(* IEC 61131-3 sources: SCLTeamCoder/experiment/datasets/oscat/oscat_code (part 4) *)

(* ---- FT_IMP.st ---- *)
FUNCTION_BLOCK FT_IMP
VAR_INPUT
    in : REAL;
    T : TIME;
    K : REAL := 1.0;
END_VAR

VAR_OUTPUT
    out : REAL;
END_VAR

VAR
    t1 : FT_PT1;
END_VAR
T1(in:= in, T:=T);
out := (in - t1.out) * K;

(*
hm 3.1.2007	rev 1.1
	added factor K

*)
END_FUNCTION_BLOCK

(* ---- FT_INT.st ---- *)
FUNCTION_BLOCK FT_INT
VAR_INPUT
    IN : REAL;
    K : REAL := 1;
    RUN : BOOL := TRUE;
    RST : BOOL;
    OUT_MIN : REAL := -1E+37;
    OUT_MAX : REAL := 1E+37;
END_VAR

VAR_OUTPUT
    OUT : REAL;
    LIM : BOOL;
END_VAR

VAR
    INTeg : INTEGRATE;
END_VAR
IF rst THEN
	out := 0.0;
ELSE
	integ(X := IN, E := RUN, K := K, Y := out);
END_IF;

(* limit the outputs *)
IF out >= OUT_MAX THEN
	out := out_max;
	LIM := TRUE;
ELSIF out <= out_min THEN
	out := out_min;
	lim := TRUE;
ELSE
	lim := FALSE;
END_IF;

(*
hm 13.12.2006	rev 1.1
	changed to "trapezregel" which increases accuracy
	before out := out + in * time new: out := out + (in + in_last) / 2 * time

hm 15.1.2007		rev 1.2
	added default for k to be 1.

hm	15.9.2007		rev 1.3
	replaced time() with T_PLC_US for compatibility and performance reason
	increased internal accuracy to microseconds

hm 29. oct 2007		rev 1.4
	changed code so int will not be called is time difference is 0 to increase accuracy on systems
	with cycle times below 1ms

hm	2. dec 2007	 	rev 1.5
	changed code for better performance

hm	5. jan 2008		rev 1.6
	further improvements in performance

hm	8. feb 2008		rev 1.7
	deleted limits +/- 1000 now limit is the range of real
	added variables out1 and out2 to extend the resolution
	corrected an error with elapsed time
	deleted unusfull output ET

hm	13. mar 2008	rev 1.8
	changed preset value out_min to -1e37.
	stop integrator at the limits.

hm	16. mar 2008	rev 1.9
	added type conversion to avoid warning under codesys 3.0

hm	2. jun. 2008	rev 2.0
	rewritten with clear code
	limits can now be set without run

hm	3. nov. 2008	rev 2.1
	optimized code using INTEGRATE and LIMX

hm	10. mar. 2009	rev 2.2
	removed nested comments
*)
END_FUNCTION_BLOCK

(* ---- FT_INT2.st ---- *)
FUNCTION_BLOCK FT_INT2
VAR_INPUT
    IN : REAL;
    K : REAL := 1.0;
    RUN : BOOL := TRUE;
    RST : BOOL;
    OUT_MIN : REAL := -1E+38;
    OUT_MAX : REAL := 1E+38;
END_VAR

VAR_OUTPUT
    OUT : REAL;
    LIM : BOOL;
END_VAR

VAR
    integ : INTEGRATE;
    ix : REAL;
    val : REAL2;
END_VAR
IF RST THEN
	val := R2_SET(0.0);
	out := 0.0;
ELSE
	integ(X := IN, E := RUN, K := K, Y := ix);
	val := R2_ADD(val, ix);
	ix := 0.0;
	OUT := val.RX;
END_IF;

(* check output for limits *)
IF out > OUT_MIN AND out < OUT_MAX THEN
	LIM := FALSE;
ELSE
	OUT := LIMIT(OUT_MIN, OUT, OUT_MAX);
	val := R2_SET(OUT);
	LIM := TRUE;
END_IF;

(*	revision history
hm	2. jun. 2008	rev 1.0
	original version

hm	5. nov. 2008	rev 1.1
	rewritten code using integrate

hm	11. mar. 2009	rev 1.2
	real constants updated to new systax using dot

*)
END_FUNCTION_BLOCK

(* ---- FT_MIN_MAX.st ---- *)
FUNCTION_BLOCK FT_MIN_MAX
VAR_INPUT
    in : REAL;
    rst : BOOL;
END_VAR

VAR_OUTPUT
    mx : REAL;
    mn : REAL;
END_VAR

VAR
    init : BOOL;
END_VAR
IF rst OR NOT init THEN
	mn := in;
	mx := in;
	init := TRUE;
ELSIF in < mn THEN mn := in;
ELSIF in > mx THEN mx := in;
END_IF;
END_FUNCTION_BLOCK

(* ---- FT_PD.st ---- *)
FUNCTION_BLOCK FT_PD
VAR_INPUT
    IN : REAL;
    KP : REAL := 1.0;
    TV : REAL := 1.0;
END_VAR

VAR_OUTPUT
    Y : REAL;
END_VAR

VAR
    diff : FT_DERIV;
END_VAR
(* run differentiator *)
diff(IN := IN, K := TV);

(* combine both values *)
Y := KP * (diff.out + IN);

(* revision history
hm 	3. jun. 2008 	rev 1.0
	original version

*)
END_FUNCTION_BLOCK

(* ---- FT_PDT1.st ---- *)
FUNCTION_BLOCK FT_PDT1
VAR_INPUT
    IN : REAL;
    KP : REAL := 1.0;
    TV : REAL := 1.0;
    T1 : REAL := 1.0;
END_VAR

VAR_OUTPUT
    Y : REAL;
END_VAR

VAR
    diff : FT_DERIV;
    TP : FT_PT1;
END_VAR
(* run differentiator *)
diff(IN := IN, K := TV);

(* Run PT1 filter *)
tp(in := diff.out, T := REAL_TO_TIME(T1));

(* combine both values *)
Y := KP * (tp.out + IN);

(* revision history
hm 	3. jun. 2008 	rev 1.0
	original version

*)
END_FUNCTION_BLOCK

(* ---- FT_PI.st ---- *)
FUNCTION_BLOCK FT_PI
VAR_IN
    IN : REAL;
    KP : REAL := 1.0;
    KI : REAL := 1.0;
    ILIM_L : REAL := -1E+38;
    ILIM_H : REAL := 1E+38;
    IEN : BOOL := TRUE;
    RST : BOOL;
END_VAR

VAR_OUT
    Y : REAL;
    LIM : BOOL;
END_VAR

VAR
    integ : FT_INT;
END_VAR
(* run integrator *)
integ(IN := IN, K := KI, RUN := IEN, RST := RST, OUT_MIN := ILIM_L, OUT_MAX := ILIM_H);

(* check if integrator has reached its limits and set overflow *)
LIM := integ.LIM;
Y := KP * IN + integ.Out;

(* revision history
hm 	3. jun. 2008 	rev 2.0
	original version

*)
END_FUNCTION_BLOCK

(* ---- FT_PID.st ---- *)
FUNCTION_BLOCK FT_PID
VAR_INPUT
    IN : REAL;
    KP : REAL := 1.0;
    TN : REAL := 1.0;
    TV : REAL := 1.0;
    ILIM_L : REAL := -1E+38;
    ILIM_H : REAL := 1E+38;
    IEN : BOOL := TRUE;
    RST : BOOL;
END_VAR

VAR_OUTPUT
    Y : REAL;
    LIM : BOOL;
END_VAR

VAR
    integ : FT_INT;
    diff : FT_DERIV;
END_VAR
(* run integrator only if TN > 0 *)
IF TN > 0.0 THEN
	integ(IN := IN, K := 1.0 / TN, RUN := IEN, RST := RST, OUT_MIN := ILIM_L, OUT_MAX := ILIM_H);
ELSE
	integ(RST := FALSE);
END_IF;

(* run differentiator *)
diff(IN := IN, K := TV);

(* combine both values *)
Y := KP * (integ.Out + diff.out + IN);

(* check if integrator has reached its limits and set overflow *)
LIM := integ.LIM;

(* revision history
hm 3. jun. 2008 	rev 2.0
	original version

hm	11. mar. 2009	rev 2.1
	real constants updated to new systax using dot

*)
END_FUNCTION_BLOCK

(* ---- FT_PIDW.st ---- *)
FUNCTION_BLOCK FT_PIDW
VAR_INPUT
    IN : REAL;
    KP : REAL := 1.0;
    TN : REAL := 1.0;
    TV : REAL := 1.0;
    LIM_L : REAL := -1E+38;
    LIM_H : REAL := 1E+38;
    RST : BOOL;
END_VAR

VAR_OUTPUT
    Y : REAL;
    LIM : BOOL;
END_VAR

VAR
    integ : INTEGRATE;
    diff : FT_DERIV;
    YI : REAL;
END_VAR
(* run the integrator *)
IF tn = 0.0 OR rst THEN
	integ(E := FALSE, Y := YI);
	YI := 0.0;
ELSE
	integ(X := IN, K := 1.0 / TN, E := NOT LIM, Y := YI);
END_IF;

(* add up integrator and linear part *)
Y := KP * (IN + YI);

(* run differentiator *)
diff(IN := IN, K := TV);

(* set lim before differentiator is added to stop integrator if necessary *)
IF Y > LIM_L AND Y < LIM_H THEN
	LIM := FALSE;
ELSE
	LIM := TRUE;
END_IF;

(* add differential part and limit output Y *)

Y := LIMIT(LIM_L, Y + KP * diff.out, LIM_H);

(* revision history
hm 3. jun. 2008 	rev 1.0
	original version

hm	5. nov. 2008	rev 1.1
	changed code to use integrate

hm	11. mar. 2009	rev 1.2
	real constants updated to new systax using dot

*)
END_FUNCTION_BLOCK

(* ---- FT_PIDWL.st ---- *)
FUNCTION_BLOCK FT_PIDWL
VAR_INPUT
    IN     : REAL;
    KP     : REAL := 1.0;
    TN     : REAL := 1.0;
    TV     : REAL := 1.0;
    LIM_L  : REAL := -1E+38;
    LIM_H  : REAL := 1E+38;
    RST    : BOOL;
END_VAR

VAR_OUTPUT
    Y      : REAL;
    LIM    : BOOL;
END_VAR

VAR
    piwl   : FT_PIWL; // derived type
    diff   : FT_DERIV; // derived type
END_VAR
(* if rst then *)
IF rst THEN
	piwl(rst := TRUE);
	piwl.RST := FALSE;
ELSE
	(* run PIWL controller first *)
	(* we need to check if TN = 0 and do alternative calls *)
	IF TN = 0.0 THEN
		piwl(in := IN * KP, KP := 1.0, KI := 0.0, LIM_L := LIM_L, LIM_H := LIM_H);
	ELSE
		piwl(in := IN * KP, KP := 1.0, KI := 1.0 / TN, LIM_L := LIM_L, LIM_H := LIM_H);
	END_IF;

	(* run differentiator and add_to_output *)
	diff(IN := IN, K := KP * TV);
	Y := piwl.Y + diff.out;

	(* limit the output *)
	IF Y < LIM_L THEN
		LIM := TRUE;
		Y := LIM_L;
	ELSIF Y > LIM_H THEN
		LIM := TRUE;
		Y := LIM_H;
	ELSE
		LIM := FALSE;
	END_IF;
END_IF;

(* revision history
hm 13. jun. 2008 	rev 1.0
	original version

hm	25. jan 2008	rev 1.1
	multiply differential part with KP

hm	11. mar. 2009	rev 1.2
	real constants updated to new systax using dot

hm	13. nov. 2009	rev 1.3
	fixed code for negative KP

*)
END_FUNCTION_BLOCK

(* ---- FT_PIW.st ---- *)
FUNCTION_BLOCK FT_PIW
VAR_INPUT
    IN : REAL;
    KP : REAL := 1.0;
    KI : REAL := 1.0;
    LIM_L : REAL := -1E+38;
    LIM_H : REAL := 1E+38;
    RST : BOOL;
END_VAR

VAR_OUTPUT
    Y : REAL;
    LIM : BOOL;
END_VAR

VAR
    integ : FT_INT;
END_VAR
(* run integrator *)
integ(IN := IN, K := KI, RUN := NOT LIM, RST := RST);

(* set output value *)
Y := KP * IN + integ.Out;

(* check for limits and set integrator for anti wind up *)
IF Y < LIM_L THEN
	Y := LIM_L;
	LIM := TRUE;
ELSIF Y > LIM_H THEN
	Y := LIM_H;
	LIM := TRUE;
ELSE
	LIM := FALSE;
END_IF;

(* revision history
hm 	3. jun. 2008 	rev 1.0
	original version

*)
END_FUNCTION_BLOCK

(* ---- FT_PIWL.st ---- *)
FUNCTION_BLOCK FT_PIWL
VAR_INPUT
    IN : REAL;
    KP : REAL := 1.0;
    KI : REAL := 1.0;
    LIM_L : REAL := -1E+38;
    LIM_H : REAL := 1E+38;
    RST : BOOL;
END_VAR

VAR_OUTPUT
    Y : REAL;
    LIM : BOOL;
END_VAR

VAR
    init : BOOL;
    tx : DWORD;
    tc : REAL;
    t_last : DWORD;
    in_last : REAL;
    i : REAL;
    p : REAL;
END_VAR
(* initialize at power_up *)
IF NOT init OR RST THEN
	init := TRUE;
	in_last := in;
	t_last := T_PLC_US();
	i := 0.0;
	tc := 0.0;
ELSE
	(* read last cycle time in Microseconds *)
	tx := T_PLC_US();
	tc := DWORD_TO_REAL(tx - t_last);
	t_last := tx;

	(* calculate proportional part *)
	p := KP * IN;

	(* run integrator *)
	i := (IN + in_last) * 5.0E-7 * KI * tc + i;
	in_last := IN;

	(* calculate output Y *)
	Y := p + i;

	(* check output for limits *)
	IF Y >= LIM_H THEN
		Y := LIM_H;
		IF ki <> 0.0 THEN
			i := LIM_H - p;
		ELSE
			i := 0.0;
		END_IF;
		LIM := TRUE;
	ELSIF Y <= LIM_L THEN
		Y := LIM_L;
		IF ki <> 0.0 THEN
			i := LIM_L - p;
		ELSE
			i := 0.0;
		END_IF;
		LIM := TRUE;
	ELSE
		LIM := FALSE;
	END_IF;
END_IF;

(* revision history
hm 13. jun. 2008 	rev 1.0
	original version

hm	27. oct. 2008	rev 1.1
	integrator will not be adjusted when ki = 0

hm	25. jan 2009	rev 1.2
	module will also work with negative K

hm	11. mar. 2009	rev 1.3
	real constants updated to new systax using dot

*)
END_FUNCTION_BLOCK

(* ---- FT_Profile.st ---- *)
FUNCTION_BLOCK FT_Profile
VAR_INPUT
    K : REAL := 1.0;
    O : REAL;
    M : REAL := 1.0;
    E : BOOL;
    value_0 : REAL;
    time_1 : TIME;
    value_1 : REAL;
    time_2 : TIME;
    value_2 : REAL;
    time_3 : TIME;
    value_3 : REAL;
    time_10 : TIME;
    value_10 : REAL;
    time_11 : TIME;
    value_11 : REAL;
    time_12 : TIME;
    value_12 : REAL;
    time_13 : TIME;
    value_13 : REAL;
END_VAR_INPUT

VAR_OUTPUT
    Y : REAL;
    RUN : BOOL;
    ET : TIME;
END_VAR_OUTPUT

VAR
    tx : TIME;
    edge : BOOL;
    state : BYTE;
    ta : TIME;
    tb : TIME;
    t0 : TIME;
    temp : REAL;
    va : REAL;
    vb : REAL;
END_VAR
(* read system time *)
tx := DWORD_TO_TIME(T_PLC_MS());

(* determine start condition *)
IF E AND NOT edge THEN
	RUN := TRUE;
	ET := t#0s;
	t0 := tx;
	ta := tx;
	tb := multime(time_1, M);
	va := value_0;
	vb := value_1;
	temp := value_0;
	state := 1;
END_IF;
edge := E;

(* generate startup profile *)
IF run THEN
	CASE state OF
		1:	IF tx - ta >= tb THEN
				ta := ta + tb;
				tb := multime(time_2 - time_1, M);
				va := value_1;
				vb := value_2;
				temp := value_1;
				state := 2;
			ELSE
				temp := ((vb - va) * TIME_TO_REAL(tx - ta) / TIME_TO_REAL(tb) + va);
			END_IF;
		2:	IF tx - ta >= tb THEN
				ta := ta + tb;
				tb := multime(time_3 - time_2, M);
				va := value_2;
				vb := value_3;
				temp := value_2;
				state := 3;
			ELSE
				temp := ((vb - va) * TIME_TO_REAL(tx - ta) / TIME_TO_REAL(tb) + va);
			END_IF;
		3:	IF tx - ta >= tb THEN
				ta := ta + tb;
				tb := multime(time_10 - time_3, M);
				va := value_3;
				vb := value_10;
				temp := value_3;
				state := 4;
			ELSE
				temp := ((vb - va) * TIME_TO_REAL(tx - ta) / TIME_TO_REAL(tb) + va);
			END_IF;
		4 :	IF tx - ta >= tb THEN
				ta := ta + tb;
				tb := multime(time_11 - time_10, M);
				va := value_10;
				vb := value_11;
				temp := value_10;
				IF E THEN state := 5; ELSE state := 6; END_IF;
			ELSE
				temp := ((vb - va) * TIME_TO_REAL(tx - ta) / TIME_TO_REAL(tb) + va);
			END_IF;
		5:	(* extend the signal while E is true *)
			IF E THEN
				ta := tx;
			ELSE
				state := 6;
			END_IF;
		6:	IF tx - ta >= tb THEN
				ta := ta + tb;
				tb := multime(time_12 - time_11, M);
				va := value_11;
				vb := value_12;
				temp := value_11;
				state := 7;
			ELSE
				temp := ((vb - va) * TIME_TO_REAL(tx - ta) / TIME_TO_REAL(tb) + va);
			END_IF;
		7:	IF tx - ta >= tb THEN
				ta := ta + tb;
				tb := multime(time_13 - time_12, M);
				va := value_12;
				vb := value_13;
				temp := value_12;
				state := 8;
			ELSE
				temp := ((vb - va) * TIME_TO_REAL(tx - ta) / TIME_TO_REAL(tb) + va);
			END_IF;
		8:	IF tx - ta >= tb THEN
				temp := value_13;
				run := FALSE;
			ELSE
				temp := ((vb - va) * TIME_TO_REAL(tx - ta) / TIME_TO_REAL(tb) + va);
			END_IF;
	END_CASE;
	Y := temp * K + O;
	ET := tx - t0;
END_IF;

(* revision history
hm	27 feb 2007		rev 1.0
	original version

hm	15. sep2007		rev 1.1
	replaced Time() with T_PLC_MS for compatibility and performance reasons

*)
END_FUNCTION_BLOCK

(* ---- FT_PT1.st ---- *)
FUNCTION_BLOCK FT_PT1
VAR_INPUT
    in : REAL;
    T : TIME;
    K : REAL := 1.0;
END_VAR

VAR_OUTPUT
    out : REAL;
END_VAR

VAR
    last : DWORD;
    tx : DWORD;
    init : BOOL;
END_VAR
(* read system time *)
tx := T_PLC_US();

(* startup initialisation *)
IF NOT init OR T = t#0s THEN
	init := TRUE;
	out := K * in;
ELSE
	out := out + (in * K - out) * DWORD_TO_REAL(Tx - last) / TIME_TO_REAL(T) * 1.0E-3;
	IF ABS(out) < 1.0E-20 THEN out := 0.0; END_IF;
END_IF;
last := tx;

(*
hm 1.1.2007	rev 1.1
	corrected error while startup value was not correct
	for very small time values real output would run out of range.

hm 3.1.2007	rev 1.2
	corrected an error for falling edge failures.
	added output faktor K.

hm 27. 2. 2007	rev 1.3
	output will be input during init for definitive startup condition.

hm	15.9.2007	rev 1.4
	changed time() to T_PLC_US() for compatibilitxy resons
	increased internal accuracy to Microseconds instead of Milliseconds

hm	23. oct 2007	rev 1.5
	added out := in to the init statements

hm	30. nov 2007	rev 1.6
	changed out to be K * in during initialization

hm	5. jan 2008	rev 1.7
	improved code for better performance

hm	16. mar. 2008	rev 1.8
	added type conversion to avoid warning under codesys 3.0

hm	14. jun. 2008	rev 1.9
	improved code

hm	11. mar. 2009	rev 1.10
	real constants updated to new systax using dot

hm	18. jan. 2011	rev 1.11
	avoid underrun of out
*)
END_FUNCTION_BLOCK

(* ---- FT_PT2.st ---- *)
FUNCTION_BLOCK FT_PT2
VAR_INPUT
    in : REAL;
    T : TIME;
    D : REAL;
    K : REAL := 1.0;
END_VAR

VAR_OUTPUT
    out : REAL;
END_VAR

VAR
    init : BOOL;
    int1 : INTEGRATE;
    int2 : INTEGRATE;
    tn : REAL;
    I1 : REAL;
    I2 : REAL;
    tn2 : REAL;
END_VAR
(* startup initialisation *)
IF NOT init OR T = T#0s THEN
	init := TRUE;
	out := K * in;
	I2 := out;
ELSE
	TN := TIME_TO_REAL(T) * 1.0E-3;
	tn2 := TN * TN;
	int1(X := in * K / tn2 - I1 * 0.5 * D / TN - I2 / TN2, Y := I1);
	int2(X := I1,Y := I2);
	out := I2;
END_IF;

(* revision history

15.1.2007 hm		rev 1.1
	changed formula to new more acurate formula

hm 15.9.2007		rev 1.2
	deleted unused code for init system time reading tx

hm	30.11.2007	rev 1.3
	changed out to be K * in during initialization
	avoind divide by 0 if tn = 0

hm	3. nov. 2008	rev 1.4
	optimized code and fixed a problem with init

hm	11. mar. 2009	rev 1.5
	real constants updated to new systax using dot

*)
END_FUNCTION_BLOCK

(* ---- FT_RMP.st ---- *)
FUNCTION_BLOCK FT_RMP
VAR_INPUT
    Rmp : BOOL := TRUE;
    in : REAL;
    KR : REAL;
    KF : REAL;
END_VAR

VAR_OUTPUT
    out : REAL;
    busy : BOOL;
    UD : BOOL;
END_VAR

VAR
    tx : TIME;
    last : TIME;
    init : BOOL;
END_VAR
(* read system time *)
tx := DWORD_TO_TIME(T_PLC_MS()) - last;

IF NOT init THEN
	init := TRUE;
	last := tx;
	tx := t#0s;
	out := in;
END_IF;
IF NOT rmp THEN
	out := in;
	busy := FALSE;
ELSIF out > in THEN
	(* ramp down *)
	out := out - TIME_TO_REAL(tx) * 0.001 * KF;
	out := MAX(in, out);
ELSIF out < in THEN
	(* ramp up *)
	out := out + TIME_TO_REAL(tx) * 0.001 * KR;
	out := MIN(in, out);
END_IF;

(* set busy and dir flags *)
IF out < in THEN
	busy := TRUE;
	ud := TRUE;
ELSIF out > in THEN
	busy := TRUE;
	ud := FALSE;
ELSE
	busy := FALSE;
END_IF;
last := last + tx;

(* revision history:

hm 8.10.2006			rev 1.1
	added ud output

hm 12. feb 2007		rev 1.2
	added init variable and corrected a possible startup problem

hm	17. sep 2007	rev 1.3
	replaced time() with t_plc_ms() for compatibility reasons

hm	25. jan 2008	rev 1.4
	performance improvements
	allow KR and KF to be 0
*)
END_FUNCTION_BLOCK

(* ---- FT_TN16.st ---- *)
FUNCTION_BLOCK FT_TN16
VAR_INPUT
    in : REAL;
    T : TIME;
END_VAR

VAR_OUTPUT
    out : REAL;
    trig : BOOL;
END_VAR

VAR
    length : INT := 16;
    X : ARRAY[0..15] OF REAL;
    cnt : INT;
    last : TIME;
    tx : TIME;
    init : BOOL;
END_VAR
(* read system time *)
tx := DWORD_TO_TIME(T_PLC_MS());

trig := FALSE;
IF NOT init THEN
	x[cnt] := in;
	init := TRUE;
	last := tx;
ELSIF tx - last >= T / length THEN
	IF cnt = length - 1 THEN cnt := 0; ELSE cnt := cnt + 1; END_IF;
	Out := X[cnt];
	x[cnt] := in;
	last := tx;
	Trig := TRUE;
END_IF;

(* revision history
hm		1. jan 2007	rev 1.0
	original version

hm		16. sep 2007	rev 1.1
	changes time() to T_plc_ms() for compatibility reasons

*)
END_FUNCTION_BLOCK

(* ---- FT_TN64.st ---- *)
FUNCTION_BLOCK FT_TN64
VAR_INPUT
    in: REAL;
    T: TIME;
END_VAR

VAR_OUTPUT
    out: REAL;
    trig: BOOL;
END_VAR

VAR
    length: INT := 64;
    X: ARRAY[0..63] OF REAL;
    cnt: INT;
    last: TIME;
    tx: TIME;
    init: BOOL;
END_VAR
(* read system time *)
tx := DWORD_TO_TIME(T_PLC_MS());

trig := FALSE;
IF NOT init THEN
	x[cnt] := in;
	init := TRUE;
	last := tx;
ELSIF tx - last >= T / length THEN
	IF cnt = length - 1 THEN cnt := 0; ELSE cnt := cnt + 1; END_IF;
	Out := X[cnt];
	x[cnt] := in;
	last := tx;
	trig := TRUE;
END_IF;

(* revision history
hm		1. jan 2007		rev 1.0
	original version

hm		16. sep 2007	rev 1.1
	changes time() to T_plc_ms() for compatibility reasons

*)
END_FUNCTION_BLOCK

(* ---- FT_TN8.st ---- *)
FUNCTION_BLOCK FT_TN8
VAR_INPUT
    in : REAL;
    T : TIME;
END_VAR

VAR_OUTPUT
    out : REAL;
    trig : BOOL;
END_VAR

VAR
    length : INT := 8;
    X : ARRAY[0..7] OF REAL;
    cnt : INT;
    last : TIME;
    tx : TIME;
    init : BOOL;
END_VAR
tx := DWORD_TO_TIME(T_PLC_MS());
trig := FALSE;
IF NOT init THEN
	x[cnt] := in;
	init := TRUE;
	last := tx;
ELSIF tx - last >= T / length THEN
	IF cnt = length - 1 THEN cnt := 0; ELSE cnt := cnt + 1; END_IF;
	Out := X[cnt];
	x[cnt] := in;
	last := tx;
	trig := TRUE;
END_IF;

(* revision history
hm		1. jan 2007		rev 1.0
	original version

hm		16. sep 2007	rev 1.1
	changes time() to T_plc_ms() for compatibility reasons

*)
END_FUNCTION_BLOCK

(* ---- GEN_BIT.st ---- *)
FUNCTION_BLOCK GEN_BIT
VAR_INPUT
    in0 : DWORD;
    in1 : DWORD;
    in2 : DWORD;
    in3 : DWORD;
    clk : BOOL;
    steps : INT;
    rep : INT;
    rst : BOOL;
END_VAR

VAR_OUTPUT
    Q0 : BOOL;
    Q1 : BOOL;
    Q2 : BOOL;
    Q3 : BOOL;
    cnt : INT;
    run : BOOL;
END_VAR

VAR
    r0 : DWORD;
    r1 : DWORD;
    r2 : DWORD;
    r3 : DWORD;
    rx : INT := 1;
END_VAR
(* check if number of runs is finished or rep = 0 which means continuous *)

IF clk AND NOT rst THEN
	run := (rep = 0) OR (rx <= rep);
	IF run THEN
		(* check for step counter reached and reset to 0 if cnt = steps *)
		IF cnt = steps THEN
			cnt := 0;
		END_IF;

		(* when cnt = 0 then reload the inputs into the registers *)
		IF cnt = 0 THEN
			r0 := in0;
			r1 := in1;
			r2 := in2;
			r3 := in3;
		END_IF;

		(* when cnt < steps, shift the lowest bits to the outputs *)
		IF (cnt < steps) THEN
			Q0 := r0.0;
			Q1 := r1.0;
			Q2 := r2.0;
			Q3 := r3.0;
			r0 := SHR(r0,1);
			r1 := SHR(r1,1);
			r2 := SHR(r2,1);
			r3 := SHR(r3,1);
		END_IF;

		(* increment the step counter *)
		cnt := cnt +1;
		IF (cnt = steps) AND (rep <> 0) THEN rx := rx +1; END_IF;
		IF (rx > rep) AND (rep <> 0) THEN run := FALSE; END_IF;
	END_IF;
ELSE
	IF rst THEN
		run := FALSE;
		Q0 := FALSE;
		Q1 := FALSE;
		Q2 := FALSE;
		Q3 := FALSE;
		r0 := 0;
		r1 := 0;
		r2 := 0;
		r3 := 0;
		cnt := 0;
		rx := 1;
	END_IF;
END_IF;

(* revision histroy
hm	4 aug 2006	rev 1.0
	original version

hm 15. oct. 2008	rev 1.1
	improved performance

hm	14. mar. 2009	rev 1.2
	removed double assignments

*)
END_FUNCTION_BLOCK

(* ---- GEN_PULSE.st ---- *)
FUNCTION_BLOCK GEN_PULSE
VAR_INPUT
    ENQ : BOOL := TRUE;
    PTH : TIME;
    PTL : TIME;
END_VAR

VAR_OUTPUT
    Q : BOOL;
END_VAR

VAR
    tx : TIME;
    tn : TIME;
    init : BOOL;
END_VAR
IF enq THEN
	tx := DWORD_TO_TIME(T_PLC_MS());
	IF NOT init THEN init := TRUE; tn := tx; END_IF;
	IF tx - tn >= SEL(Q, PTL, PTH) THEN
		tn := tn + SEL(Q, PTL, PTH);
		Q := NOT Q;
	END_IF;
ELSE
	Q := FALSE;
	init := FALSE;
END_IF;

(* revision history
hm	29. jun. 2008	rev 1.0
	original version

hm	23. nov. 2008	rev 1.1
	set default for enq to be true

hm	18. jul. 2009	rev 1.2
	improved performance

hm	13. nov. 2009	rev 1.3
	corrected error

hm	16. feb. 2011	rev 1.4
	corrected an error when timer overflows

hm	8. apr. 2011	rev 1.5
	ptl and pth was exchanged
*)
END_FUNCTION_BLOCK

(* ---- GEN_PW2.st ---- *)
FUNCTION_BLOCK GEN_PW2
VAR_INPUT
    ENQ: BOOL;
    TH1: TIME;
    TL1: TIME;
    TH2: TIME;
    TL2: TIME;
    TS: BOOL;
END_VAR

VAR_OUTPUT
    Q: BOOL;
    TH: TIME;
    TL: TIME;
END_VAR

VAR
    t_high: TIME;
    t_low: TIME;
    tx: TIME;
    start: TIME;
    init: BOOL;
    et: TIME;
END_VAR
(* read system timer *)
tx := DWORD_TO_TIME(T_PLC_MS());

(* startup initialization *)
IF NOT init THEN
	start := tx;
	init := TRUE;
	TH := T#0s;
	TL := T#0s;
END_IF;

(* timing selection *)
IF TS THEN
	t_high := TH2;
	t_low := TL2;
ELSE
	t_high := TH1;
	t_low := TL1;
END_IF;

(* normal operation *)
IF ENQ THEN
	et := tx - start;
	IF NOT Q THEN
		IF et >= t_low THEN
			Q := TRUE;
			start := tx;
			TL := T#0s;
		ELSE
			TL := et;
		END_IF;
	ELSE
		IF et >= t_high THEN
			Q := FALSE;
			start := tx;
			TH := T#0s;
		ELSE
			TH := et;
		END_IF;
	END_IF;
ELSE
	Q := FALSE;
	TH := T#0s;
	TL := T#0s;
	start := tx;
END_IF;

(* revision history
hm	26. sep. 2008	rev 1.0
	original version

hm	14. mar. 2009	rev 1.1
	removed double assignments

*)
END_FUNCTION_BLOCK

(* ---- GEN_RDM.st ---- *)
FUNCTION_BLOCK GEN_RDM
VAR_INPUT
    PT : TIME;
    AM : REAL := 1;
    OS : REAL;
END_VAR

VAR_OUTPUT
    Q : BOOL;
    Out : REAL;
END_VAR

VAR
    tx : TIME;
    last : TIME;
    init : BOOL;
END_VAR
(* read system time and prepare input data *)
tx := DWORD_TO_TIME(T_PLC_MS()) - last;

(* init section *)
IF NOT init THEN
	init := TRUE;
	last := tx;
	tx := t#0s;
END_IF;

(* add last if one cycle is finished *)
IF tx >= pt THEN
	last := last + pt;
	tx := tx - pt;

	(* generate output signal *)
	out := am * (RDM(0) - 0.5) + os;
	q := TRUE;
ELSE
	q := FALSE;
END_IF;

(* revision history

hm	7.2.2007		rev 1.0
	original version

hm	16.9.2007		rev 1.1
	changes time() to T_plc_ms() for compatibility reasons

*)
END_FUNCTION_BLOCK

(* ---- GEN_RDT.st ---- *)
FUNCTION_BLOCK GEN_RDT
VAR_INPUT
    Enable : BOOL := TRUE;
    Min_Time_ms : TIME := TIME#1s0ms; // min Taktzeit
    Max_Time_ms : TIME := TIME#1s200ms; // Max Taktzeit
    TP_Q : TIME := TIME#100ms; // Zeit Ausgang auf TRUE
END_VAR

VAR_OUTPUT
    xQ : BOOL;
END_VAR

VAR
    tonRDMTimer : TON; // Zeitbaustein Taktgenerator
    tof_xQ : TOF; // Ausschaltverzögerung Taktgenerator
    tRDMTime : TIME; // Sollzeit
    rRDMTime : REAL; // Zufalswert Timer
END_VAR
tonRDMTimer ( IN:= Enable , PT:= tRDMTime );
tof_xQ ( IN:= tonRDMTimer.Q , PT:= TP_Q );
XQ := tof_xq.Q;
IF tonRDMTimer.Q THEN
		 xQ := TRUE ;
		 rRDMTime := RDM ( last:= rRDMTime ) ;
		 tRDMTime := REAL_TO_TIME ( rRDMTime * DINT_TO_REAL(TIME_TO_DINT( Max_Time_ms - Min_Time_ms ) + TIME_TO_DINT(Min_Time_ms ))) ;
		 tonRDMTimer ( IN:= FALSE );
END_IF;

(* revision history
J. Schohaus	19. nov 2007	rev 1.0
	origial version

hm	16. mar. 2008			rev 1.1
	added type conversion to avoid warnings under codesys 3.0
*)
END_FUNCTION_BLOCK

(* ---- GEN_RMP.st ---- *)
FUNCTION_BLOCK GEN_RMP
VAR_INPUT
    PT : TIME := TIME#1s0ms;
    AM : REAL := 1.0;
    OS : REAL;
    DL : REAL;
END_VAR

VAR_OUTPUT
    Q : BOOL;
    OUT : REAL;
END_VAR

VAR
    tx : TIME;
    last : TIME;
    init : BOOL;
    temp : REAL;
    ltemp : REAL;
END_VAR
(* read system time and prepare input data *)
tx := DWORD_TO_TIME(T_PLC_MS()) - last;
DL := MODR(dl,1.0);
IF dl < 0.0 THEN dl := 1.0 - dl; END_IF;

(* init section *)
IF NOT init THEN
	init := TRUE;
	last := tx;
	tx := t#0s;
END_IF;

(* add last if one cycle is finished *)
IF tx >= pt THEN
	last := last + pt;
	tx := tx - pt;
END_IF;

(* generate sine wave *)
ltemp := temp;
IF pt > t#0s THEN temp := FRACT(TIME_TO_REAL(tx + MULTIME(pt, dl)) / TIME_TO_REAL(pt)); END_IF;
out := am * temp + os;

(* boolean output Q *)
Q := temp < ltemp;

(* revision history
hm	3. mar 2007		rev 1.0
	original version

hm	17 sep 2007		rev 1.1
	replaced time() with t_plc_ms for compatibilitx reasons

hm	27. nov 2007	rev 1.2
	avoid divide by 0 when pt = 0

ks	26. oct. 2008	rev 1.3
	code optimization

hm	10. mar. 2009	rev 1.4
	changed real constants to use dot syntax
*)
END_FUNCTION_BLOCK

(* ---- GEN_SIN.st ---- *)
FUNCTION_BLOCK GEN_SIN
VAR_INPUT
    PT : TIME;
    AM : REAL := 1.0;
    OS : REAL;
    DL : REAL;
END_VAR

VAR_OUTPUT
    Q : BOOL;
    Out : REAL;
END_VAR

VAR
    tx : TIME;
    last : TIME;
    init : BOOL;
    temp : REAL;
END_VAR
(* read system time and prepare input data *)
tx := DWORD_TO_TIME(T_PLC_MS()) - last;
DL := MODR(dl,1.0);
IF dl < 0.0 THEN dl := 1.0 - dl; END_IF;

(* init section *)
IF NOT init THEN
	init := TRUE;
	last := tx;
	tx := t#0s;
END_IF;

(* add last if one cycle is finished *)
IF tx >= pt THEN
	last := last + pt;
	tx := tx - pt;
END_IF;

(* generate sine wave *)
IF pt > t#0s THEN temp := SIN(math.PI2 * DWORD_TO_REAL(TIME_TO_DWORD(tx + MULTIME(pt, dl))) / DWORD_TO_REAL(TIME_TO_DWORD(pt))); END_IF;
out := am * 0.5 *  temp + os;

(* boolean output Q *)
q := NOT SIGN_R(temp);

(* revision history
hm	22. jan 2007	rev 1.0
	original version

hm	17 sep 2007	rev 1.1
	replaced time() with t_plc_ms for compatibilitx reasons

hm	27. nov 2007	rev 1.2
	avoid divide by 0 when pt = 0

hm	6. jan 2008		rev 1.3
	improved performance

hm	16. mar. 2008	rev 1.4
	added type conversion to avoid warnings under codesys 3.0

hm	18. oct. 2008	rev 1.5
	using math constants

hm	11. mar. 2009	rev 1.6
	changed real constants to use dot syntax

*)
END_FUNCTION_BLOCK

(* ---- GEN_SQ.st ---- *)
FUNCTION_BLOCK GEN_SQ
VAR_INPUT
    PT: TIME;
END_VAR

VAR_OUTPUT
    Q: BOOL;
END_VAR

VAR
    tn: DWORD;
    tx: DWORD;
    init: BOOL;
END_VAR
(* read system time *)
tx := T_PLC_MS();

IF NOT init THEN
	init := TRUE;
	tn := tx;
	Q := TRUE;
ELSIF tx - tn >= SHR(TIME_TO_DWORD(PT),1) THEN
	Q := NOT Q;
	tn := tn + SHR(TIME_TO_DWORD(pt),1);
END_IF;

(* revision history
hm	4. aug 2006	rev 1.0
	original version

hm	17. sep 2007	rev 1.1
	replaced time() with T_PLC_MS() for compatibility reasons

hm	18. jul. 2009	rev 1.2
	improved accuracy

hm	16. feb 2011	rev 1.3
	corrected an error with timer overflow
*)
END_FUNCTION_BLOCK

(* ---- GEN_SQR.st ---- *)
FUNCTION_BLOCK GEN_SQR
VAR_INPUT
    PT : TIME;
    AM : REAL := 1.0;
    OS : REAL;
    DC : REAL := 0.5;
    DL : REAL;
END_VAR

VAR_OUTPUT
    Q : BOOL;
    Out : REAL;
END_VAR

VAR
    tx : TIME;
    last : TIME;
    init : BOOL;
END_VAR
(* check dc = 1 or 0 *)
IF dc = 0.0 THEN
	out := -am * 0.5 + os;
	Q := FALSE;
	RETURN;
ELSIF dc = 1.0 THEN
	out := am * 0.5 + os;
	Q := TRUE;
	RETURN;
END_IF;

(* read system time and prepare input data *)
tx := DWORD_TO_TIME(T_PLC_MS()) - last;
DL := MODR(dl,1.0);
IF dl < 0.0 THEN dl := 1.0 - dl; END_IF;
dc := MODR(dc,1.0);
IF dc < 0.0 THEN dc := 1.0 - dc; END_IF;

(* init section *)
IF NOT init THEN
	init := TRUE;
	last := tx;
	tx := t#0s;
END_IF;

(* add last if one cycle is finished *)
IF tx >= pt THEN
	last := last + pt;
	tx := tx - pt;
END_IF;

(* check if falling or rising edge first *)
IF MULTIME(pt, dl + dc) >= pt THEN
	(* generate falling edge *)
	IF tx >= MULTIME(pt, dl + dc - 1) THEN
		out := -am * 0.5 + os;
		Q := FALSE;
	END_IF;
	(* generate rising edge *)
	IF tx >= MULTIME(pt, dl) THEN
		out := am * 0.5 + os;
		Q := TRUE;
	END_IF;
ELSE
	(* generate rising edge first *)
	IF tx >= MULTIME(pt, dl) THEN
		out := am * 0.5 + os;
		Q := TRUE;
	END_IF;
	(* generate falling edge *)
	IF tx >= MULTIME(pt, dl + dc) THEN
		out := -am * 0.5 +os;
		Q := FALSE;
	END_IF;
END_IF;

(* revision history

hm	12. feb 2007	rev 1.1
	added default value for dc = 0.5

hm	17 sep 2007	rev 1.2
	replaced time() with t_plc_ms for compatibilitx reasons

hm	6. jan 2008	rev 1.3
	improved performance

hm	11. mar. 2009	rev 1.4
	changed real constants to use dot syntax
	set default amplitude to 1.0

*)
END_FUNCTION_BLOCK

(* ---- HOLIDAY.st ---- *)
FUNCTION_BLOCK HOLIDAY
VAR_INPUT
    DATE_IN : DATE;
    LANGU : INT;
    FRIDAY : BOOL;
    SATURDAY : BOOL;
    SUNDAY : BOOL;
END_VAR_INPUT

VAR_IN_OUT
    HOLIDAYS : ARRAY[0..29] OF HOLIDAY_DATA;
END_VAR_IN_OUT

VAR CONSTANT
    SIZE : INT := 29;
END_VAR CONSTANT

VAR_OUTPUT
    Y : BOOL;
    NAME : STRING[30];
END_VAR_OUTPUT

VAR
    last_active : DATE;
    ostern : DATE;
    i : INT;
    jahr : INT;
    x_date : DATE;
    lx : INT;
    wdx : INT;
END_VAR
(* for performance reasons only activate once a day *)
IF last_active = date_in THEN RETURN; END_IF;
last_active := DATE_IN;

(* determine language *)
IF LANGU = 0 THEN
	lx := language.DEFAULT;
ELSE
	lx := MIN(language.LMAX, LANGU);
END_IF;

(* berechnung von ostern für das aktuelle jahr *)
jahr := YEAR_OF_DATE(date_in);
ostern := EASTER(jahr);
wdx := DAY_OF_WEEK(DATE_IN);
Y := FALSE;

(* check for holidays *)
FOR i := 0 TO size DO
	x_date := SET_DATE(jahr, HOLIDAYS[i].MONTH , HOLIDAYS[i].DAY);
	IF HOLIDAYS[i].USE = 1 AND HOLIDAYS[i].MONTH > 0 THEN
		(* check for fixed date holiday *)
		IF x_date = date_in THEN
			Y := TRUE;
			NAME := HOLIDAYS[i].NAME;
			RETURN;
		END_IF;
	ELSIF HOLIDAYS[i].USE = 1 AND HOLIDAYS[i].MONTH = 0 THEN
		(* check for holiday in reference to easter *)
		IF DATE_ADD(ostern, HOLIDAYS[i].DAY ,0,0,0) = date_in THEN
			Y := TRUE;
			NAME := HOLIDAYS[i].NAME;
			RETURN;
		END_IF;
	ELSIF HOLIDAYS[i].USE < 0 THEN
		(* check for holiday on a weekday before date *)
		IF DAY_OF_WEEK(date_in) = ABS(HOLIDAYS[i].USE) AND date_in < x_date AND date_in >= DATE_ADD(x_date,-7,0,0,0) THEN
			Y := TRUE;
			NAME := HOLIDAYS[i].NAME;
			RETURN;
		END_IF;
	END_IF;
END_FOR;

(* check array if today is weekend *)
IF NOT Y AND (wdx = 5 AND FRIDAY OR wdx = 6 AND SATURDAY OR wdx = 7 AND SUNDAY) THEN
	Y := TRUE;
	NAME := LANGUAGE.WEEKDAYS[LOCATION.LANGUAGE[lx],wdx];
ELSE
	NAME := '';
END_IF;

(*
Neujahrstag 	1. Januar 	• 	• 	• 	• 	• 	• 	• 	• 	• 	• 	• 	• 	• 	• 	• 	•
Heilige Drei Könige 	6. Januar 	• 	• 												•
Karfreitag 	Ostersonntag - 2d 	• 	• 	• 	• 	• 	• 	• 	• 	• 	• 	• 	• 	• 	• 	• 	•
Ostersonntag 	siehe Osterdatum 				(•)
Ostermontag 	Ostersonntag + 1d 	• 	• 	• 	• 	• 	• 	• 	• 	• 	• 	• 	• 	• 	• 	• 	•
Tag der Arbeit 	1. Mai 	• 	• 	• 	• 	• 	• 	• 	• 	• 	• 	• 	• 	• 	• 	• 	•
Christi Himmelfahrt 	Ostersonntag + 39d 	• 	• 	• 	• 	• 	• 	• 	• 	• 	• 	• 	• 	• 	• 	• 	•
Pfingstsonntag 	Ostersonntag + 49d 				(•)
Pfingstmontag 	Ostersonntag + 50d 	• 	• 	• 	• 	• 	• 	• 	• 	• 	• 	• 	• 	• 	• 	• 	•
Fronleichnam 	Ostersonntag + 60d 	• 	• 					• 			• 	• 	• 	1) 			2)
Augsburger Friedensfest 	8. August 		(3)
Mariä Himmelfahrt 	15. August 		(5) 										•
Tag der Deutschen Einheit 	3. Oktober 6) 	• 	• 	• 	• 	• 	• 	• 	• 	• 	• 	• 	• 	• 	• 	• 	•
Reformationstag 	31. Oktober 				• 				• 					• 	• 		•
Allerheiligen 	1. November 	• 	• 								• 	• 	•
Buß- und Bettag 4) 	Mittwoch vor dem 23.11. 			7 										•
1. Weihnachtstag 	25. Dezember 	• 	• 	• 	• 	• 	• 	• 	• 	• 	• 	• 	• 	• 	• 	• 	•
2. Weihnachtstag 	26. Dezember 	• 	• 	• 	• 	• 	• 	• 	• 	• 	• 	• 	• 	• 	• 	• 	•
*)

(* revision history
hm 	27. feb. 2007	rev 1.1
	deleted unused variable init

hm	31. oct. 2007	rev 1.2
	changed holiday definition from constant to input constant to allow easier changes by user without recompilation of the lib

hm 	24. nov. 2007	rev 1.3
	changes F_use of  Buß_und_Bettag to 0 because this is no official holiday

hm	7. apr. 2008	rev 1.4
	improved performance

hm	7. oct. 2008	rev 1.5
	changed code to use setup data from global constants
	changed length of output NAME from 20 to 30
	holiday will now also be indicated on a weekend
	changed function year to year_of_date
	changed function weekday to day_of_week

hm	21. oct. 2008	rev 1.6
	using location constants

hm	18. jan 2011	rev 2.0
	using user specified array for holidays

*)
END_FUNCTION_BLOCK

(* ---- HYST.st ---- *)
FUNCTION_BLOCK HYST
VAR_INPUT
    In : REAL;
    ON : REAL;
    OFF : REAL;
END_VAR

VAR_OUTPUT
    Q : BOOL;
    win : BOOL;
END_VAR
IF ON >= OFF THEN
	IF IN < OFF THEN
		Q := FALSE;
		WIN := FALSE;
	ELSIF  IN > ON THEN
		Q := TRUE;
		WIN := FALSE;
	ELSE
		WIN := TRUE;
	END_IF;
ELSE
	IF IN > OFF THEN
		Q := FALSE;
		WIN := FALSE;
	ELSIF  IN < ON THEN
		Q := TRUE;
		WIN := FALSE;
	ELSE
		WIN := TRUE;
	END_IF;
END_IF;

(* revision history
hm		2.  jun 2008	rev 1.0
	original version

*)
END_FUNCTION_BLOCK

(* ---- HYST_1.st ---- *)
FUNCTION_BLOCK HYST_1
VAR_INPUT
    In : REAL;
    high : REAL;
    low : REAL;
END_VAR_INPUT

VAR_OUTPUT
    Q : BOOL;
    win : BOOL;
END_VAR_OUTPUT
IF in < low THEN
	Q := FALSE;
	win := FALSE;
ELSIF in > high THEN
	Q := TRUE;
	win := FALSE;
ELSE
	win := TRUE;
END_IF;

(* revision history
hm		4.  aug. 2006	rev 1.0
	original version

hm		2. jun. 2008	rev 1.1
	improved performance
*)
END_FUNCTION_BLOCK

(* ---- HYST_2.st ---- *)
FUNCTION_BLOCK HYST_2
VAR_INPUT
    IN   : REAL;
    VAL  : REAL;
    HYS  : REAL;
END_VAR

VAR_OUTPUT
    Q    : BOOL;
    WIN  : BOOL;
END_VAR

VAR
    tmp  : REAL;
END_VAR
tmp := val - hys * 0.5;
IF in < tmp THEN
	Q := FALSE;
	win := FALSE;
ELSIF in > tmp + hys THEN
	Q := TRUE;
	win := FALSE;
ELSE
	win := TRUE;
END_IF;

(* revision history
hm		4. aug 2006	rev 1.0
	original version

hm		5. jan 2008	rev 1.1
	improved code for better performance

hm		2. jun. 2008	rev 1.2
	improved performance
*)
END_FUNCTION_BLOCK

(* ---- HYST_3.st ---- *)
FUNCTION_BLOCK HYST_3
VAR_INPUT
    in : REAL;
    hyst : REAL;
    val1 : REAL;
    val2 : REAL;
END_VAR

VAR_OUTPUT
    Q1 : BOOL;
    Q2 : BOOL;
END_VAR

VAR
    X : REAL;
END_VAR
X := hyst * 0.5;
IF in < val1 - X THEN
	q1 := TRUE;
ELSIF in > val1 + X THEN
	q1 := FALSE;
END_IF;
IF in < val2 - X THEN
	q2 := FALSE;
ELSIF in > val2 + X THEN
	q2 := TRUE;
END_IF;

(* revision history
hm	22. jan 2007	rev 1.0
	original version

hm	27. dec 2007	rev 1.1
	changed code for better performance

hm	5. jan 2008	rev 1.2
	further performance iprovements

*)
END_FUNCTION_BLOCK

(* ---- INC_DEC.st ---- *)
FUNCTION_BLOCK INC_DEC
VAR_INPUT
    CHa : BOOL;
    CHb : BOOL;
    RST : BOOL;
END_VAR

VAR_OUTPUT
    dir : BOOL;
    cnt : INT;
END_VAR

VAR
    edgea : BOOL;
    clk : BOOL;
    clka : BOOL;
    clkb : BOOL;
    edgeb : BOOL;
    axb : BOOL;
END_VAR
axb := cha XOR chb;

(* create pulses for channel a *)
clka := cha XOR edgea;
edgea := cha;

clkb := chb XOR edgeb;
edgeb := chb;

(* create pulses for both channels *)
clk := clka OR clkb;

(* set the direction output *)
IF axb AND clka THEN dir := TRUE; END_IF;
IF axb AND clkb THEN dir := FALSE; END_IF;

(* increment or decrement the counter *)
IF clk AND dir THEN cnt := cnt + 1; END_IF;
IF clk AND NOT dir THEN cnt := cnt -1; END_IF;

(* reset the counter if rst active *)
IF rst THEN cnt := 0; END_IF;
END_FUNCTION_BLOCK

(* ---- INTEGRATE.st ---- *)
FUNCTION_BLOCK INTEGRATE
VAR_INPUT
    E : BOOL := TRUE;
    X : REAL;
    K : REAL := 1.0;
END_VAR

VAR_IN_OUT
    Y : REAL;
END_VAR

VAR
    X_last : REAL;
    init : BOOL;
    last : DWORD;
    tx : DWORD;
END_VAR
(*read system time *)
tx := T_PLC_MS();

IF NOT init THEN
	init := TRUE;
	X_last := X;
ELSIF E THEN
	Y := (X + X_LAST) * 0.5E-3 * DWORD_TO_REAL(tx-last) * K + Y;
	X_last := X;
END_IF;
last := tx;

(*
hm 3. nov. 2008	rev 1.0
original version

*)
END_FUNCTION_BLOCK

(* ---- INTERLOCK.st ---- *)
FUNCTION_BLOCK INTERLOCK
VAR_INPUT
    I1: BOOL;
    I2: BOOL;
    TL: TIME;
END_VAR

VAR_OUTPUT
    Q1: BOOL;
    Q2: BOOL;
END_VAR

VAR
    T1: TON; (* Assuming TOF is implemented as a derivative needs - please replace with appropriate declaration if different *)
    T2: TON; (* Assuming TOF is implemented as a derivative needs - please replace with appropriate declaration if different *)
END_VAR
(* the input signal have a run delay to lockout the other input *)
T1(IN := I1, PT := TL);
T2(IN := I2, PT := TL);

Q1 := I1 AND NOT t2.Q;
Q2 := I2 AND NOT t1.Q;

(* revision history

hm	28 sep 2007		rev 1.0
	original version

*)
END_FUNCTION_BLOCK

(* ---- INTERLOCK_4.st ---- *)
FUNCTION_BLOCK INTERLOCK_4
VAR_INPUT
    I0 : BOOL;
    I1 : BOOL;
    I2 : BOOL;
    I3 : BOOL;
    E : BOOL;
    MODE : INT;
END_VAR

VAR_OUTPUT
    OUT : BYTE;
    TP : BOOL;
END_VAR

VAR
    in : BYTE;
    last : BYTE;
    old : BYTE;
    lmode : INT;
END_VAR
(* check if enable is active *)
IF E THEN
(* reset all vars when there is a mode change on thy fly *)
	IF mode <> lmode THEN
		out := 0;
		last := 0;
		old := 0;
		lmode := mode;
	END_IF;
	(* load inputs into in *)
	in.0 := I0;
	in.1 := I1;
	in.2 := I2;
	in.3 := I3;
	(* only execute when there is any change *)
	IF in <> last THEN
		(* only execute when inputs have chages state *)
		CASE mode OF
			0:	(* output directly display inputs as bits in byte out *)
				out := in;

			1:	(* the input with the highest number will be acepted *)
				IF in.3 THEN out := 8;
				ELSIF in.2 THEN out := 4;
				ELSIF in.1 THEN out := 2;
				ELSE out := in;
				END_IF;

			2:	(* input last pressed will be displayed only *)
				last := ((in XOR last) AND in);
				IF last.3 THEN out := 8;
				ELSIF last.2 THEN out := 4;
				ELSIF last.1 THEN out := 2;
				ELSE out := last;
				END_IF;

			3:	(* any input active will disable all other inputs *)
				IF (out AND in) = 0 THEN
					IF in.3 THEN out := 8;
					ELSIF in.2 THEN out := 4;
					ELSIF in.1 THEN out := 2;
					ELSE out := in;
					END_IF;
				END_IF;

		END_CASE;
		last := in;
	END_IF;
	tp := out <> old;
	old := out;
ELSE
	out := 0;
	last := 0;
	old := 0;
	lmode := 0;
	tp := FALSE;
END_IF;

(* revision history
hm	24. oct 2008	rev 1.0
	original version

hm	14. mar. 2009	rev 1.1
	replaced double assignments

*)
END_FUNCTION_BLOCK

(* ---- LENGTH.st ---- *)
FUNCTION_BLOCK LENGTH
VAR_INPUT
    m : REAL;
    p : REAL;
    in : REAL;
    ft : REAL;
    yd : REAL;
    mile : REAL;
    sm : REAL;
    fm : REAL;
END_VAR

VAR_OUTPUT
    Ym : REAL;
    Yp : REAL;
    Yin : REAL;
    Yft : REAL;
    Yyd : REAL;
    Ymile : REAL;
    Ysm : REAL;
    Yfm : REAL;
END_VAR
Ym :=	m
		+ p * 0.000376065
		+ in * 0.0254
		+ ft * 0.3048
		+ yd * 0.9144
		+ mile * 1609.344
		+ sm * 1852.0
		+ fm * 1.829;
Yp := Ym * 2659.11478068951;
Yin := Ym * 39.37007874016;
Yft := Ym * 3.28083989501;
Yyd := Ym * 1.09361329834;
Ymile := Ym * 0.00062137119;
Ysm := Ym * 0.00053995680;
Yfm := Ym * 0.54674685621;

(*
Länge Meter m SI-Basiseinheit
Astronomische Einheit* AE 1 AE = 149,597 870 · E9 m
Parsec pc 1 pc = 206265 AE = 30,857 · E15 m
Lichtjahr Lj 1 Lj = 9,460 530 · E15 m = 63240 AE = 0,306 59 pc
Ångström Å 1 Å = E–l0 m
typograph. Punkt p 1 p = 0,376 065 mm • im Druckereigewerbe
inch** in 1 in = 2,54 · E–2 m = 25,4 mm***
foot ft 1 ft = 0,3048 m = 30,48 cm
yard yd 1 yd = 0,9144 m
mile mile 1 mile = 1609,344 m
Internat. Seemeile sm 1 sm = 1852 m
Fathom fm 1 fm = 1,829 m • in der Seeschifffahrt
*)

(* revision history

hm	27. mar. 2007	rev 1.0
	original version

hm	11. mar. 2009	rev 1.1
	improved code

*)
END_FUNCTION_BLOCK

(* ---- LIST_NEXT.st ---- *)
FUNCTION_BLOCK LIST_NEXT
VAR_INPUT
    SEP : BYTE;
    RST : BOOL;
END_VAR

VAR_IN_OUT
    LIST : STRING(LIST_LENGTH);
END_VAR_IN_OUT

VAR_OUTPUT
    LEL : STRING(LIST_LENGTH);
    NUL : BOOL;
END_VAR_OUTPUT

VAR
    pos : INT := 1;
    pt : POINTER TO ARRAY[1..LIST_LENGTH] OF BYTE;
    po : POINTER TO ARRAY[1..LIST_LENGTH] OF BYTE;
    c : BYTE;
    write : INT;
END_VAR
pt := ADR(LIST);
po := ADR(LEL);

IF rst THEN
	pos := 1;
END_IF;

IF pt^[pos] = 0 OR pos = LIST_LENGTH THEN
	LEL := '';
	NUL := TRUE;
ELSE
	NUL := FALSE;
	write := 1;
	FOR pos := pos + 1 TO LIST_LENGTH DO
		c := pt^[pos];
		IF c = 0 OR c = SEP THEN
			po^[write] := 0;
			RETURN;
		ELSE
			po^[write] := pt^[pos];
			write := write + 1;
		END_IF;
	END_FOR;
END_IF;

(* revision histroy
hm	25. jun. 2008	rev 1.0
	original release

hm	19. jan. 2011	rev 1.1
	changed string(255) to string(LIST_LENGTH)

hm	21. mar. 2011	rev 2.0
	all elements start with SEP

*)
END_FUNCTION_BLOCK

(* ---- LTCH.st ---- *)
FUNCTION_BLOCK LTCH
VAR_INPUT
    D : BOOL;
    L : BOOL;
    RST : BOOL;
END_VAR

VAR_OUTPUT
    Q : BOOL;
END_VAR
(* as long as L is true, the latch is transparent and and change of D is transferred to Q *)
(* of course only when there is no asynchronous reset *)
IF rst THEN				(* if asynchronous reset then Q=0 *)
	Q := FALSE;
ELSIF L THEN			(* latch is transparent *)
	Q := D;
END_IF;

(* revision history
hm	4. aug 2006		rev 1.0
	original version

hm	27. dec 2007	rev 1.1
	changed code for better performance

hm	30. oct. 2008	rev 1.2
	deleted unnecessary init with 0

*)
END_FUNCTION_BLOCK

(* ---- LTCH_4.st ---- *)
FUNCTION_BLOCK LTCH_4
VAR_INPUT
    D0 : BOOL;
    D1 : BOOL;
    D2 : BOOL;
    D3 : BOOL;
    L  : BOOL;
    RST : BOOL;
END_VAR

VAR_OUTPUT
    Q0 : BOOL;
    Q1 : BOOL;
    Q2 : BOOL;
    Q3 : BOOL;
END_VAR
(* as long as L is true, the latch is transparent and and change of D is transferred to Q *)
(* of course only when there is no asynchronous reset *)
IF rst THEN			(* if asynchronous reset then Q=0 *)
	Q0 := FALSE;
	Q1 := FALSE;
	Q2 := FALSE;
	Q3 := FALSE;
ELSIF L THEN			(* latch is transparent *)
	Q0 := D0;
	Q1 := D1;
	Q2 := D2;
	Q3 := D3;
END_IF;

(* revision history
hm	4. aug 2006	rev 1.0
	original version

hm	27. dec 2007	rev 1.1
	changed code for better performance

hm	30. oct. 2008	rev 1.2
	deleted unnecessary init with 0

hm	14. mar. 2009	rev 1.3
	removed double assignments

*)
END_FUNCTION_BLOCK

(* ---- M_D.st ---- *)
FUNCTION_BLOCK M_D
VAR_INPUT
    start : BOOL;
    stop : BOOL;
    tmax : TIME := TIME#14400m0s0ms;
    rst : BOOL;
END_VAR

VAR_OUTPUT
    PT : TIME;
    ET : TIME;
    run : BOOL;
END_VAR

VAR
    edge : BOOL;
    T0 : TIME;
    tx : TIME;
    startup : BOOL;
END_VAR
(* check for rst input *)
IF rst OR et >= tmax THEN
	pt := t#0ms;
	et := t#0ms;
	startup := FALSE;
	run := FALSE;
END_IF;

(* avoid timers to start when input is true at startup *)
IF NOT startup THEN
	edge := start;
	startup := TRUE;
END_IF;

(* read system timer *)
tx := DWORD_TO_TIME(T_PLC_MS());

(* detect rising edge on start *)
IF start AND NOT edge AND NOT stop THEN
	t0 := tx;
	run := TRUE;
	pt := t#0s;
ELSIF stop AND run THEN
	pt := et;
	run := FALSE;
END_IF;
edge := start;
IF run THEN et := tx - t0; END_IF;

(* revision history
hm		2.5.2007	rev 1.0
	original version

hm		16.9.2007	rev 1.1
	changes time() to T_plc_ms() for compatibility reasons

hm	27. feb 2009	rev 1.2
	deleted unnecessary init with 0
*)
END_FUNCTION_BLOCK

(* ---- M_T.st ---- *)
FUNCTION_BLOCK M_T
VAR_INPUT
    IN : BOOL;
    TMAX : TIME := TIME#14400m0s0ms;
    RST : BOOL;
END_VAR

VAR_OUTPUT
    PT : TIME;
    ET : TIME;
END_VAR

VAR
    edge : BOOL;
    start : TIME;
    tx : TIME;
END_VAR
(* read system time *)
tx := DWORD_TO_TIME(T_PLC_MS());

IF RST OR ET >= TMAX THEN
	PT :=  t#0s;
	ET := t#0s;
ELSIF IN THEN
	IF NOT edge THEN start := tx; END_IF;
	ET := tx - start;
ELSE
	PT := ET;
END_IF;
edge := IN;

(* revision history
hm	4. aug. 2006	rev 1.0
	original version

hm	2. may. 2007	rev 1.1
	added init variable to avoid unreasonable measurement if falling edge occurs first.
	added et (elapsed time) output to count from 0 at rising edge until a falling edge resets et to 0.
	added reset input.

hm	16. sep. 2007	rev 1.2
	changes time() to T_plc_ms() for compatibility reasons

hm	17. dec. 2008	rev 1.3
	code optimized

hm	10. mar. 2009	rev 1.4
	removed nested comments
	removed double assignments

*)
END_FUNCTION_BLOCK

(* ---- M_TX.st ---- *)
FUNCTION_BLOCK M_TX
VAR_INPUT
    in : BOOL;
    tmax : TIME := TIME#14400m0s0ms;
    rst : BOOL;
END_VAR

VAR_OUTPUT
    TH : TIME;
    TL : TIME;
    DC : REAL;
    F : REAL;
    ET : TIME;
END_VAR

VAR
    edge : BOOL;
    start : TIME;
    stop : TIME;
    tx : TIME;
    rise : BOOL;
    fall : BOOL;
    startup : BOOL;
END_VAR
(* check FOR rst input *)
IF rst OR (et >= tmax) THEN
	rise := FALSE;
	fall := FALSE;
	startup := FALSE;
	th := t#0ms;
	tl := t#0ms;
	DC := 0.0;
	F := 0.0;
	ET := t#0s;
END_IF;

(* avoid timers to start when input is true at startup *)
IF NOT startup THEN
	edge := in;
	startup := TRUE;
END_IF;

(* read system timer *)
tx := DWORD_TO_TIME(T_PLC_MS());

(* edge trigger rising and falling edge *)
IF in XOR edge THEN
	edge := in;
	(* rising edge starts measurement *)
	IF in THEN
		start := Tx;
		rise := TRUE;
		IF fall THEN tl := start - stop; END_IF;
		IF th > t#0ms AND tl > t#0ms THEN
			dc := TIME_TO_REAL(th) / TIME_TO_REAL(th+tl);
			f := 1000.0 / TIME_TO_REAL(th + tl);
		END_IF;
	(* falling edge starts second cycle measurement *)
	ELSE
		stop := Tx;
		fall := TRUE;
		IF rise THEN th := stop - start; END_IF;
		IF th > t#0ms AND tl > t#0ms THEN
			dc := TIME_TO_REAL(th) /  TIME_TO_REAL(th+tl);
			f := 1000.0 / TIME_TO_REAL(th + tl);
		END_IF;
	END_IF;
END_IF;
IF rise THEN et := tx - start; END_IF;

(* revision history
hm	4. aug. 2006	rev 1.0
	original version

hm	2. mai. 2007	rev 1.1
	made sure that no undefined values would be measured at startup conditions
	added output et
	added rst input
	added tmax input

hm	16. sep. 2007	rev 1.2
	changes time() to T_plc_ms() for compatibility reasons

hm	27. feb. 2009	rev 1.3
	deleted unnecessary init with 0

hm	11. mar. 2009	rev 1.4
	changed real constants to use dot syntax

*)
END_FUNCTION_BLOCK

(* ---- MANUAL_1.st ---- *)
FUNCTION_BLOCK MANUAL_1
VAR_INPUT
    IN : BOOL;
    MAN : BOOL;
    M_I : BOOL;
    SET : BOOL;
    RST : BOOL;
END_VAR

VAR_OUTPUT
    Q : BOOL;
    STATUS : BYTE;
END_VAR

VAR
    S_edge : BOOL;
    r_edge : BOOL;
    edge : BOOL;
END_VAR
IF NOT man THEN
	Q := IN;
	STATUS := 100;
	edge := FALSE;
ELSIF NOT s_edge AND set THEN
	Q := TRUE;
	edge := TRUE;
	status := 101;
ELSIF NOT r_edge AND rst THEN
	Q := FALSE;
	edge := TRUE;
	status := 102;
ELSIF NOT edge THEN
	Q := M_I;
	status := 103;
END_IF;

(* remember levels of manual signals *)
s_edge := SET;
r_edge := RST;

(* revision history
hm	17. jun 2008	rev 1.0
	original version

hm	17. oct 2008	rev 1.1
	deleted unnecessary variable m_edge

hm	14. mar. 2009	rev 1.2
	replaced double assignments

*)
END_FUNCTION_BLOCK

(* ---- MANUAL_2.st ---- *)
FUNCTION_BLOCK MANUAL_2
VAR_INPUT
    IN : BOOL;
    ENA : BOOL;
    ON : BOOL;
    OFF : BOOL;
    MAN : BOOL;
END_VAR

VAR_OUTPUT
    Q : BOOL;
    STATUS : BYTE;
END_VAR
IF ena THEN
	IF NOT ON AND NOT OFF THEN
		Q := IN;
		STATUS := 100;
	ELSIF on AND NOT off THEN
		Q := TRUE;
		STATUS := 101;
	ELSIF NOT on AND off THEN
		q := FALSE;
		STATUS := 102;
	ELSE
		Q := MAN;
		STATUS := 103;
	END_IF;
ELSE
	Q := FALSE;
	STATUS := 104;
END_IF;

(* revision history
hm	22. sep. 2008		rev 1.0
	original version

*)
END_FUNCTION_BLOCK

(* ---- MANUAL_4.st ---- *)
FUNCTION_BLOCK MANUAL_4
VAR_INPUT
    I0 : BOOL;
    I1 : BOOL;
    I2 : BOOL;
    I3 : BOOL;
    MAN : BOOL;
    STP : BOOL;
    M0 : BOOL;
    M1 : BOOL;
    M2 : BOOL;
    M3 : BOOL;
END_VAR

VAR_OUTPUT
    Q0 : BOOL;
    Q1 : BOOL;
    Q2 : BOOL;
    Q3 : BOOL;
    STATUS : BYTE;
END_VAR

VAR
    edge : BOOL;
    pos : INT;
    tog : BOOL;
END_VAR
IF man THEN
	IF NOT TOG THEN
		Q0 := M0;
		Q1 := M1;
		Q2 := M2;
		Q3 := M3;
		STATUS := 101;
	END_IF;
	IF STP AND NOT edge THEN
		tog := TRUE;
		CASE pos OF
			0:	Q0 := TRUE;
				Q1 := FALSE;
				Q2 := FALSE;
				Q3 := FALSE;
				STATUS := 110;
			1:	Q0 := FALSE;
				Q1 := TRUE;
				Q2 := FALSE;
				Q3 := FALSE;
				STATUS := 111;
			2:	Q0 := FALSE;
				Q1 := FALSE;
				Q2 := TRUE;
				Q3 := FALSE;
				STATUS := 112;
			3:	Q0 := FALSE;
				Q1 := FALSE;
				Q2 := FALSE;
				Q3 := TRUE;
				STATUS := 113;
		END_CASE;
		pos := INC(pos,1,3);
	END_IF;
ELSE
	Q0 := I0;
	Q1 := I1;
	Q2 := I2;
	Q3 := I3;
	STATUS := 100;
	tog := FALSE;
	pos := 0;
END_IF;

(* remember status of stp *)
edge := STP;

(* revision history
hm	17. jun 2008		rev 1.0
	original version

*)
END_FUNCTION_BLOCK

(* ---- MATRIX.st ---- *)
FUNCTION_BLOCK MATRIX
VAR_INPUT
    x1 : BOOL;
    x2 : BOOL;
    x3 : BOOL;
    x4 : BOOL;
    X5 : BOOL;
    Release : BOOL; (* input_constant *)
END_VAR_INPUT

VAR_OUTPUT
    code : BYTE;
    TP : BOOL;
    y1 : BOOL := TRUE;
    y2 : BOOL;
    y3 : BOOL;
    y4 : BOOL;
END_VAR_OUTPUT

VAR
    line : BYTE;
    X : ARRAY[0..3] OF BYTE; (* scan line inputs *)
    L : ARRAY[0..3] OF BYTE; (* scan line status *)
    i : INT;
    temp : BYTE;
END_VAR
TP := FALSE;
CODE := 0;
(* read scan lines *)
X[line].0 := X1;
X[line].1 := X2;
X[line].2 := X3;
X[line].3 := X4;
X[line].4 := X5;

(* compare for change *)
FOR i := 0 TO 3 DO
	IF X[i] <> L[i] THEN
		(* scan line information has changed code need to be found and generated *)
		temp := x[i] XOR L[i];
		IF temp.0 THEN
			CODE := 1;
			code.7 := X[i].0;
			L[i].0 := X[i].0;
		ELSIF temp.1 THEN
			code := 2;
			code.7 := X[i].1;
			L[i].1 := X[i].1;
		ELSIF temp.2 THEN
			code := 3;
			code.7 := X[i].2;
			L[i].2 := X[i].2;
		ELSIF temp.3 THEN
			CODE := 4;
			CODE.7 := X[i].3;
			L[i].3 := X[i].3;
		ELSIF temp.4 THEN
			CODE := 5;
			CODE.7 := X[i].4;
			L[i].4 := X[i].4;
		END_IF;
		TP := TRUE;
		CODE.4 := Line.0;
		CODE.5 := Line.1;
		CODE.6 := Line.2;

		(* check if release codes need to be killed *)
		IF NOT release AND CODE < 127 THEN
			CODE := 0;
			TP := FALSE;
		END_IF;
		EXIT;
	END_IF;
END_FOR;

(* increment scan line every cycle *)
line := (line + 1) AND 2#0000_0011;
temp := SHL(BYTE#1,line);
Y1 := temp.0;
Y2 := temp.1;
Y3 := temp.2;
Y4 := temp.3;

(* revision history
hm		10.6.2007	rev 1.0
	original version

hm		11.9.2007	rev 1.1
	deleted unused variables k and old_code

hm		23.12.2007	rev 1.2
	added exit statement in for loop instead of i:=5

hm		26. oct. 2008	rev 1.3
	code optimized

*)
END_FUNCTION_BLOCK

(* ---- MESSAGE_4R.st ---- *)
FUNCTION_BLOCK MESSAGE_4R
VAR_INPUT
    M0 : STRING(STRING_LENGTH);
    M1 : STRING(STRING_LENGTH);
    M2 : STRING(STRING_LENGTH);
    M3 : STRING(STRING_LENGTH);
    MM : INT := 3;
    ENQ : BOOL := TRUE;
    CLK : BOOL := TRUE;
    T1 : TIME := T#3s0ms;
END_VAR

VAR_OUTPUT
    MX : STRING(STRING_LENGTH);
    MN : INT;
    TR : BOOL;
END_VAR

VAR
    timer : TON;
    edge : BOOL;
END_VAR
(* check for rising edge on EN *)
TR := FALSE;
IF ENQ THEN
	IF (NOT edge AND clk) OR timer.q THEN
			MN := INC1(MN, MM);
			TR := TRUE;
			timer(in := FALSE);
			CASE MN OF
				0 : MX := M0;
				1 : MX := M1;
				2 : MX := M2;
				3 : MX := M3;
			END_CASE;
	END_IF;
	edge := clk;
	timer( in := CLK, pt := T1);
ELSE
	MX := '';
	MN := 0;
END_IF;

(* revision history
hm	8. oct. 2008	rev 1.0
	original version

hm	27. oct. 2008	rev 1.1
	changed _INC to INC1

*)
END_FUNCTION_BLOCK

(* ---- MESSAGE_8.st ---- *)
FUNCTION_BLOCK MESSAGE_8
VAR_INPUT
    IN1 : BOOL;
    IN2 : BOOL;
    IN3 : BOOL;
    IN4 : BOOL;
    IN5 : BOOL;
    IN6 : BOOL;
    IN7 : BOOL;
    IN8 : BOOL;
    S1 : STRING[STRING_LENGTH];
    S2 : STRING[STRING_LENGTH];
    S3 : STRING[STRING_LENGTH];
    S4 : STRING[STRING_LENGTH];
    S5 : STRING[STRING_LENGTH];
    S6 : STRING[STRING_LENGTH];
    S7 : STRING[STRING_LENGTH];
    S8 : STRING[STRING_LENGTH];
END_VAR

VAR_OUTPUT
    M : STRING[STRING_LENGTH];
END_VAR
(* check if an alarm is present if yes set the output M otherwise clear M *)
IF in1 THEN
	M := S1;
ELSIF in2 THEN
	M := S2;
ELSIF in3 THEN
	M := S3;
ELSIF in4 THEN
	M := S4;
ELSIF in5 THEN
	M := S5;
ELSIF in6 THEN
	M := S6;
ELSIF in7 THEN
	M := S7;
ELSIF in8 THEN
	M := S8;
ELSE
	M := '';
END_IF;

(* revision history
hm	26.12.2007		rev 1.0
	original version

hm	29. mar. 2008	rev 1.1
	changed STRING to STRING(STRING_LENGTH)
*)
END_FUNCTION_BLOCK

(* ---- METER.st ---- *)
FUNCTION_BLOCK METER
VAR_INPUT
    M1 : REAL;
    M2 : REAL;
    I1 : BOOL;
    I2 : BOOL;
    D : REAL := 1.0;
    RST : BOOL;
END_VAR

VAR_IN_OUT
    MX : REAL;
END_VAR_IN_OUT

VAR
    MR : REAL; (* Derived type REAL2 assumed to be REAL *)
    MX1 : REAL; (* Current consumption value on M1 and M2 *)
    MX2 : REAL; (* Current consumption value on M1 and M2 *)
    tx : DWORD;
    last : DWORD;
    tc : REAL;
    init : BOOL;
END_VAR
(* measure the last cycle time and make sure we onle execute once every millisecond *)
tx := T_PLC_MS();
IF NOT init THEN
	init := TRUE;
	last := tx;
	mr.RX := mx;
	mr.R1 := 0.0;
ELSIF tx = last THEN
	RETURN;
ELSE
	tc := DWORD_TO_REAL(tx - last) * 0.001;
END_IF;
last := tx;

(* reset *)
IF rst THEN
	mr.R1 := 0.0;
	mr.RX := 0.0;
ELSE
	(* current consumption measurement *)
	IF I1 THEN MX1 := M1; ELSE MX1 := 0.0; END_IF;
	IF I2 THEN MX2 := M2; ELSE MX2 := 0.0; END_IF;
	(* add up the current values in a double real *)
	MR := R2_ADD(MR,(SEL(I1,0.0,mx1) + SEL(I2, 0.0, mx2)) / D * TC);
	(* set the current output value *)
	MX := mr.RX;
END_IF;

(* revision history

hm	16. sep.2007		rev 1.0
	original version

hm	7. feb 2008		rev 1.1
	use new version of ft_int to avoid a counting stop at high values
	deleted unnecessary limits

hm	24. mar. 2008	rev 1.2
	use data_type real2 to extend accuracy to 15 digits total
	do not use ft_int which adds unnecessary overhead

hm	8. feb. 2009	rev 1.3
	changed mx to be I/O
	make sure calculation works for cycle times < 1 ms

hm	8. mar. 2009	rev 1.4
	last was not updated
	code improvements

*)
END_FUNCTION_BLOCK

(* ---- METER_STAT.st ---- *)
FUNCTION_BLOCK METER_STAT
VAR_INPUT
    IN : REAL;
    DI : DATE;
    RST : BOOL;
END_VAR

VAR_IN_OUT
    Last_Day : REAL;
    Current_Day : REAL;
    Last_Week : REAL;
    Current_Week : REAL;
    Last_Month : REAL;
    Current_Month : REAL;
    Last_Year : REAL;
    Current_Year : REAL;
END_VAR

VAR RETAIN
    Year_Start : REAL;
    Month_Start : REAL;
    Week_Start : REAL;
    Day_Start : REAL;
    last_run : DATE;
END_VAR
IF rst THEN
	Last_Day := 0.0;
	Current_Day := 0.0;
	Day_start := IN;
	Last_week := 0.0;
	Current_week := 0.0;
	Week_start := in;
	Last_month := 0.0;
	Current_month := 0.0;
	month_start := in;
	last_year := 0.0;
	current_year := 0.0;
	year_start := in;
ELSE
	Current_Day := IN - Day_Start;
	Current_Week := In - Week_Start;
	Current_Month := IN - Month_Start;
	Current_Year := IN - Year_Start;
END_IF;

IF YEAR_OF_DATE(DI) > YEAR_OF_DATE(last_run) THEN
	(* a new year has started *)
	last_year := current_year;
	current_year := 0.0;
	year_start := in;
	last_month := current_month;
	current_month := 0.0;
	month_start := in;
	last_day := current_day;
	current_day := 0.0;
	day_start := in;
ELSIF MONTH_OF_DATE(DI) > MONTH_OF_DATE(last_run) THEN
	(* a new month has started, january is alrerady done by year change *)
	last_month := current_month;
	current_month := 0.0;
	month_start := in;
	last_day := current_day;
	current_day := 0.0;
	day_start := in;
ELSIF DAY_OF_YEAR(di) > DAY_OF_YEAR(last_run) THEN
	(* day has chaged, first day of year and first day of month has already been taken care of *)
	last_day := current_day;
	current_day := 0.0;
	day_start := in;
END_IF;
IF DAY_OF_WEEK(DI) < DAY_OF_WEEK(last_run) THEN
	(* a new week has started *)
	last_week := current_week;
	current_week := 0.0;
	week_start := in;
END_IF;
last_run := di;

(* revision history
hm	16. sep. 2007	rev 1.0
	original version

hm	7. oct. 2008	rev 1.1
	changed function year_to_year_of_date
	changed function month to month_of_date
	changed function weekday to day_of_week

hm	11. mar. 2009	rev 1.2
	changed real constants to use dot syntax

hm	18. jul. 2009	rev 1.3
	changes all outputs to be I/O
*)
END_FUNCTION_BLOCK

(* ---- ONTIME.st ---- *)
FUNCTION_BLOCK ONTIME
VAR_INPUT
    IN : BOOL;
    RST : BOOL;
END_VAR_INPUT

VAR_IN_OUT
    SECONDS : UDINT;
    CYCLES : UDINT;
END_VAR_IN_OUT

VAR
    tx : DWORD;
    last : DWORD;
    edge : BOOL;
    init : BOOL;
    ms : DWORD;
END_VAR
(* read system time *)
tx := T_PLC_MS();

(* make sure the first cycle works correctly *)
IF NOT init THEN
	init := TRUE;
	last := tx;
	ms := 0;
END_IF;
IF RST THEN
	SECONDS := 0;
	CYCLES := 0;
	last := tx;
	ms := 0;
ELSIF IN THEN
	(* add the current milliseconds *)
	ms := (tx - last) + ms;
	IF ms >= 1000 THEN
		seconds := seconds + 1;
		ms := ms - 1000;
	END_IF;
	cycles := cycles + BOOL_TO_UINT(NOT edge);
END_IF;
last := tx;
edge := in;

(* revision history
hm 22.2.2007		rev 1.1
	changed VAR RETAIN PERSISTENT to VAR RETAIN for better compatibility
	wago lon contollers do not support persisitent

hm 2.8.2007		rev 1.2
	adding time up in a real number will automatically lead to the point where
	small time scales like the cycle time will be below the resolution of real and therefore
	ontime would not increase in small steps as necessary
	the time is now measured internally in two  dwords and be converted to real only for
	output purposes.
	deleted the variable power because it was unnecessary

hm	16.9.2007		rev 1.3
	changes time() to T_plc_ms() for compatibility reasons

hm	2. dec. 2007	rev 1.4
	chaged code for better performance

hm	16. mar. 2008	rev 1.5
	added type conversions to avoid warnings under codesys 3.0

hm	21. oct. 2008	rev 2.0
	changed module for much better performance and allow for external result storage

hm	10. nov. 2008	rev 2.1
	increased internal resolution to milliseconds

hm	16. nov. 2008	rev 2.2
	changed typecast to avoid warnings

hm	17. dec. 2008	rev 2.3
	fixed an error when in would be true for more then 49 days

hm	17. jan 2011	rev 2.4
	init will not clear seconds and cycles, only rst clears these values

hm	18. mar. 2011	rev 2.5
	reset was not working

*)
END_FUNCTION_BLOCK

(* ---- PARSET.st ---- *)
FUNCTION_BLOCK PARSET
VAR_INPUT
    A0 : BOOL;
    A1 : BOOL;
    X01 : REAL;
    X02 : REAL;
    X03 : REAL;
    X04 : REAL;
    X11 : REAL;
    X12 : REAL;
    X13 : REAL;
    X14 : REAL;
    X21 : REAL;
    X22 : REAL;
    X23 : REAL;
    X24 : REAL;
    X31 : REAL;
    X32 : REAL;
    X33 : REAL;
    X34 : REAL;
    TC : TIME;
END_VAR

VAR_OUTPUT
    P1 : REAL;
    P2 : REAL;
    P3 : REAL;
    P4 : REAL;
END_VAR

VAR
    X : ARRAY[0..3, 1..4] OF REAL;
    S1 : REAL;
    S2 : REAL;
    S3 : REAL;
    S4 : REAL;
    tx : DWORD;
    last : DWORD;
    start : BOOL;
    set : BYTE;
    init : BOOL;
END_VAR
(* read system_time *)
tx := T_PLC_MS();

(* init sequence *)
IF NOT init THEN
	set.0 := NOT A0;
	init := TRUE;
	X[0,1] := X01;
	X[0,2] := X02;
	X[0,3] := X03;
	X[0,4] := X04;
	X[1,1] := X11;
	X[1,2] := X12;
	X[1,3] := X13;
	X[1,4] := X14;
	X[2,1] := X21;
	X[2,2] := X22;
	X[2,3] := X23;
	X[2,4] := X24;
	X[3,1] := X31;
	X[3,2] := X32;
	X[3,3] := X33;
	X[3,4] := X34;
	P1 := X01;
	P2 := X02;
	P3 := X03;
	P4 := X04;
END_IF;

(* check for input change *)
IF (A0 XOR set.0) OR (A1 XOR set.1) THEN
	(* a new set is selected *)
	set.0 := A0;
	set.1 := A1;
	IF tc > t#0s THEN
		start := TRUE;
		last := tx;
		(* save the step speed for the output changes in S *)
		S1 := (X[set,1] - P1)/DWORD_TO_REAL(TIME_TO_DWORD(tc));
		S2 := (X[set,2] - P2)/DWORD_TO_REAL(TIME_TO_DWORD(tc));
		S3 := (X[set,3] - P3)/DWORD_TO_REAL(TIME_TO_DWORD(tc));
		S4 := (X[set,4] - P4)/DWORD_TO_REAL(TIME_TO_DWORD(tc));
	END_IF;
ELSIF start AND tx - last < TIME_TO_DWORD(tc) THEN
	(* ramp the outputs to the new value *)
	P1 := X[set,1] - S1 * DWORD_TO_REAL(TIME_TO_DWORD(Tc) - tx + last);
	P2 := X[set,2] - S2 * DWORD_TO_REAL(TIME_TO_DWORD(Tc) - tx + last);
	P3 := X[set,3] - S3 * DWORD_TO_REAL(TIME_TO_DWORD(Tc) - tx + last);
	P4 := X[set,4] - S4 * DWORD_TO_REAL(TIME_TO_DWORD(Tc) - tx + last);
ELSE
	(* make sure outputs match the correct set values *)
	start := FALSE;
	P1 := X[set,1];
	P2 := X[set,2];
	P3 := X[set,3];
	P4 := X[set,4];
END_IF;

(* revision history
hm	2.11.2007		rev 1.0
	original version

hm	16. mar. 2008	rev 1.1
	added type conversions to avoid warnings under codesys 3.0

*)
END_FUNCTION_BLOCK

(* ---- PARSET2.st ---- *)
FUNCTION_BLOCK PARSET2
VAR_INPUT
    X : REAL;
    X01 : REAL;
    X02 : REAL;
    X03 : REAL;
    X04 : REAL;
    X11 : REAL;
    X12 : REAL;
    X13 : REAL;
    X14 : REAL;
    X21 : REAL;
    X22 : REAL;
    X23 : REAL;
    X24 : REAL;
    X31 : REAL;
    X32 : REAL;
    X33 : REAL;
    X34 : REAL;
    L1 : REAL;
    L2 : REAL;
    L3 : REAL;
    TC : TIME;
END_VAR

VAR_OUTPUT
    P1 : REAL;
    P2 : REAL;
    P3 : REAL;
    P4 : REAL;
END_VAR

VAR
    Pset : parset;  // assuming 'parset' is a valid type defined elsewhere
    init : BOOL;
END_VAR
(* init sequence *)
IF NOT init THEN
	init := TRUE;
	pset(TC:=TC, X01:=X01, X02:=X02, X03:=X03, X04:=X04, X11:=X11, X12:=X12, X13:=X13, X14:=X14, X21:=X21, X22:=X22, X23:=X23, X24:=X24, X31:=X31, X32:=X32, X33:=X33, X34:=X34);
END_IF;
IF ABS(X) < L1 THEN
	pset(A0 := FALSE, A1 := FALSE);
ELSIF ABS(X) < L2 THEN
	pset(A0 := TRUE, A1 := FALSE);
ELSIF ABS(x) < L3 THEN
	pset(A0 := FALSE, A1 := TRUE);
ELSE
	pset(A0 := TRUE, A1 := TRUE);
END_IF;
P1 := pset.P1;
P2 := pset.P2;
P3 := pset.P3;
P4 := pset.P4;

(* revision history
hm		3.11.2007		rev 1.0
	original version

*)
END_FUNCTION_BLOCK

(* ---- PIN_CODE.st ---- *)
FUNCTION_BLOCK PIN_CODE
VAR_INPUT
    CB : BYTE;
    E : BOOL;
    PIN : STRING[8]; // input_constant attribute is ignored in ST declaration
END_VAR

VAR_OUTPUT
    TP : BOOL;
END_VAR

VAR
    POS : INT := 1; // Initialized to 1
END_VAR
tp := FALSE;
IF e THEN
	IF CB = CODE(pin, pos) THEN
		pos := pos + 1;
		IF pos > LEN(PIN) THEN
			(* proper code is detected *)
			TP := TRUE;
			pos := 1;
		END_IF;
	ELSE
		pos := 1;
	END_IF;
END_IF;

(* revision history
hm	30. oct. 2008	rev 1.0
	original version

*)
END_FUNCTION_BLOCK

(* ---- PRESSURE.st ---- *)
FUNCTION_BLOCK PRESSURE
VAR_INPUT
    mws : REAL;
    torr : REAL;
    att : REAL;
    atm : REAL;
    pa : REAL;
    bar : REAL;
END_VAR

VAR_OUTPUT
    Ymws : REAL;
    Ytorr : REAL;
    Yatt : REAL;
    Yatm : REAL;
    Ypa : REAL;
    Ybar : REAL;
END_VAR
Ybar := bar +
		pa * 1.0E-5 +
		0.980665 * att +
		1.01325 * atm +
		0.001333224 * torr +
		0.0980665 * mws;
Ymws := ybar * 10.1971621297793;
Ytorr := ybar * 750.0615050434140;
Yatt := ybar * 1.0197162129779;
yatm := ybar * 0.9869232667160;
Ypa := ybar * 100000.0;

(*
Druck, Pascal Pa 1 Pa = 1 N/m2 = 1 kg/(s2 E m) . 0,75 E 10.2 mmHg
mechanische 1 MPa = 1 N/mm2 . fur Festigkeitsangaben
Spannung Bar bar 1 bar = 105 Pa = 103 mbar = 105 kg/(s2 E m)
Millimeter- mmHg 1 mmHg = 133,322 Pa = 1,333 22 mbar
Quecksilbersaule . nur in Heilkunde zulassig
physik. Atmosphare atm 1 atm = 1,013 25 bar
techn. Atmosphare at 1 at = 1 kp/cm2 = 0,980665 bar
Torr Torr 1 Torr = (101325/760) Pa = 1,333224 mbar
Meter-Wassersaule mWS 1 mWS = 9806,65 Pa = 98,0665 mbar
psi lbf/in2 1 lbf/in2 = 68,947 57 mbar = 6894,757 Pa

*)

(* revision history

hm	27. mar. 2007	rev 1.0
	original version

hm	11. mar. 2009	rev 1.1
	improved code

*)
END_FUNCTION_BLOCK

(* ---- PWM_DC.st ---- *)
FUNCTION_BLOCK PWM_DC
VAR_INPUT
    F : REAL;
    DC : REAL;
END_VAR

VAR_OUTPUT
    Q : BOOL;
END_VAR

VAR
    clk : CLK_PRG;
    pulse : TP_X;
    tmp : REAL;
END_VAR
IF F > 0.0 THEN
	tmp := 1000.0 / F;
	CLK(PT := REAL_TO_TIME(tmp));
	Pulse(in := clk.Q, pt := REAL_TO_TIME(tmp * DC));
	Q := pulse.Q;
END_IF;

(* revision history

hm	25. feb 2007	rev 1.1
	recoded in st for better performance and better portability

hm	27. nov 2007	rev 1.2
	avoid divide by 0 when F = 0

hm	19. oct. 2008	rev 1.3
	changed type TP_R to TP_X because of name change
	improved performance

hm	11. mar. 2009	rev 1.4
	changed real constants to use dot syntax

*)
END_FUNCTION_BLOCK

(* ---- PWM_PW.st ---- *)
FUNCTION_BLOCK PWM_PW
VAR_INPUT
    F : REAL;
    PW : TIME;
END_VAR

VAR_OUTPUT
    Q : BOOL;
END_VAR

VAR
    clk : CLK_PRG;
    pulse : TP_X;
END_VAR
IF F > 0.0 THEN
	CLK(PT := REAL_TO_TIME(1000.0 / F));
	Pulse(in := clk.Q, pt := pw);
	Q := pulse.Q;
END_IF;

(* revision history

hm	25. feb 2007	rev 1.1
	recoded in st for better performance and better portability

hm	27. nov 2007	rev 1.2
	avoid divide by 0 when F = 0

hm	9. dec 2007		rev 1.3
	corrected an error with F = 0

hm	19. oct. 2008	rev 1.4
	changed type tp_r to TP_x brecause of name change

hm	11. mar. 2009	rev 1.5
	changed real constants to use dot syntax

*)
END_FUNCTION_BLOCK

(* ---- RMP_B.st ---- *)
FUNCTION_BLOCK RMP_B
VAR_INPUT
    SET : BOOL;
    PT : TIME;
    E : BOOL := TRUE;
    UP : BOOL := TRUE;
    RST : BOOL;
END_VAR

VAR_OUTPUT
    OUT : BYTE;
    BUSY : BOOL;
    HIGH : BOOL;
    LOW : BOOL;
END_VAR

VAR
    rmp : _RMP_B;
END_VAR
(* generate ramp *)
rmp(dir := UP, E := E, TR := PT, rmp := out);

(* set or reset operation *)
IF RST THEN
	out := 0;
ELSIF SET THEN
	out := 255;
END_IF;

(* checks for outputs stable and reset or set busy flag *)
low := out = 0;
high := out = 255;
busy := NOT (low OR high) AND E;

(* revision history

hm 5.10.2006	rev 1.1
	added busy output
hm 17.1.2007	rev 1.2
	renamed input ud to up for better usability
	deleted unused variable step

hm	17.9.2007		rev 1.3
	replaced time() with t_plc_ms() for compatibility reasons

hm	28. sep 2007	rev 1.4
	added outputs on and off
	busy is now disabled while en is false
	new coding for higher accuracy and performance

hm	5. oct 2007	rev 1.5
	added statements to allow for PT to be t#0s output jumps to max or min immediately

hm	25. dec 2007	rev 1.6
	improved code for better performance

hm	16. oct. 2008	rev 1.7
	improved code for better performance

hm	18. oct. 2008	rev 1.8
	added type conversion to avoid warnings
	changed input en to e for compatibility reasons

hm	23. oct. 2008	REV 	2.0
	new code using _RMP_B

*)
END_FUNCTION_BLOCK

(* ---- RMP_SOFT.st ---- *)
FUNCTION_BLOCK RMP_SOFT
VAR_INPUT
    IN      : BOOL;
    VAL     : BYTE;
    PT_ON   : TIME;
    PT_OFF  : TIME;
END_VAR

VAR_OUTPUT
    OUT     : BYTE;
END_VAR

VAR
    rmp     : _RMP_B;
    tmp     : BYTE;
END_VAR
tmp := SEL(in, 0, val);
IF tmp > out THEN
	(* we need to ramp down *)
	rmp(dir := TRUE, E := TRUE, TR := PT_ON, rmp := out);
	(* make sure out does not surpass tmp *)
	out := MIN(out, tmp);
ELSIF tmp < out THEN
	(* we need to ramp up *)
	rmp(dir := FALSE, E := TRUE, TR := PT_OFF, rmp := out);
	(* make sure out does not surpass tmp *)
	out := MAX(out, tmp);
ELSE
	(* no ramp necessary *)
	rmp(E := FALSE, rmp := out);
END_IF;

(* revision history

hm 22.1.2007	rev 1.1
	deleted unused variables X1 and I, X2 and X3

hm	17.9.2007	rev 1.2
	replaced time() with t_plc_ms() for compatibility reasons

hm	26. oct. 2008	2.0
	new code using _rmp_b
*)
END_FUNCTION_BLOCK

(* ---- RMP_W.st ---- *)
FUNCTION_BLOCK RMP_W
VAR_INPUT
    SET : BOOL;
    PT : TIME;
    E : BOOL := TRUE;
    UP : BOOL := TRUE;
    RST : BOOL;
END_VAR_INPUT

VAR_OUTPUT
    out : WORD;
    busy : BOOL;
    high : BOOL;
    low : BOOL;
END_VAR_OUTPUT

VAR
    rmp : _RMP_W;
END_VAR
(* generate ramp *)
rmp(dir := UP, E := E, TR := PT, rmp := out);

(* set or reset operation *)
IF RST THEN
	out := 0;
ELSIF SET THEN
	out := 65535;
END_IF;

(* checks for outputs stable and reset or set busy flag *)
low := out = 0;
high := out = 65535;
busy := NOT (low OR high) AND E;

(* revision history:

hm 4.10.2006		rev 1.1
	added the busy output which signals that the ramp is running.

hm 22.1.2007		rev 1.2
	deleted unused variable step

hm	17.9.2007		rev 1.3
	replaced time() with t_plc_ms() for compatibility reasons

hm	28. sep 2007	rev 1.4
	added outputs on and off
	busy is now disabled while en is false
	new coding for higher accuracy and performance

hm	5. oct 2007	rev 1.5
	added statements to allow for PT to be t#0s output jumps to max or min immediately

hm	2. dec 2007	rev 1.6
	corrected an error in calculation of step response

hm	25. dec 2007	rev 1.7
	corrected an error while step response was too slow for fast rise times

hm	16. oct. 2008	rev 1.8
	improved performance

hm	18. oct. 2008	rev 1.9
	renamed inout EN to E for compatibility reasons

hm	23. oct. 2008	rev 2.0
	new code using _RMP_W
*)
END_FUNCTION_BLOCK

(* ---- RTC_2.st ---- *)
FUNCTION_BLOCK RTC_2
VAR_INPUT
    SET     : BOOL;
    SDT     : DT;
    SMS     : INT;
    DEN     : BOOL;
    OFS     : INT;
END_VAR

VAR_OUTPUT
    UDT     : DT;
    LOCAL_DT : DT;
    DSO     : BOOL;
    XMS     : INT;
END_VAR

VAR
    RT      : RTC_MS; (* Derived type *)
END_VAR
(* call rtc *)
RT(SET := SET, SDT := SDT, SMS := SMS);
UDT := rt.xdt;
XMS := rt.XMS;

(* check for daylight savings time and set dso output *)
DSO := DST(udt) AND DEN;

(* calculate time offset and set ldt output *)
LOCAL_DT := DWORD_TO_DT(DT_TO_DWORD(UDT) + INT_TO_DWORD(ofs + BOOL_TO_INT(DSO)*60) * 60);

(* revision history
hm		20. jan. 2008	rev 1.0
	original version

hm		20. feb. 2008	rev 1.1
	added Millisecond Set input

hm		12. jun. 2008	rev 1.2
	improved performance

hm		20. jan. 2011	rev 1.3
	changed offset to be in minutes

hm		27. apr. 2011	rev 1.4
	fixed error with local time calculation

hm     3. Feb 2021     rev 1.5
     changed LDT to LOCAL_DT for compatibility with IEC61131-3

*)
END_FUNCTION_BLOCK

(* ---- RTC_MS.st ---- *)
FUNCTION_BLOCK RTC_MS
VAR_INPUT
    SET : BOOL;
    SDT : DT;
    SMS : INT;
END_VAR

VAR_OUTPUT
    XDT : DT;
    XMS : INT;
END_VAR

VAR
    init : BOOL;
    last : DWORD;
    Tx : DWORD;
END_VAR
tx := T_PLC_MS();
IF set OR NOT init THEN
	(* clock needs to be set when set is true or after power up *)
	init := TRUE;
	xdt := SDT;
	XMS := SMS;
ELSE
	XMS := XMS + DWORD_TO_INT(tx - last);
	(* check if one second has expired *)
	IF XMS > 999 THEN
		XDT := XDT + T#1s;
		XMS := XMS - 1000;
	END_IF;
END_IF;
last := tx;

(* revision history
hm		20. jan. 2008	rev 1.0
	original version

hm		20. feb. 2008	rev 1.1
	added Millisecond Set input
*)
END_FUNCTION_BLOCK

(* ---- SCHEDULER.st ---- *)
FUNCTION_BLOCK SCHEDULER
VAR_INPUT
    E0 : BOOL;
    E1 : BOOL;
    E2 : BOOL;
    E3 : BOOL;
    T0 : TIME;
    T1 : TIME;
    T2 : TIME;
    T3 : TIME;
END_VAR

VAR_OUTPUT
    Q0 : BOOL;
    Q1 : BOOL;
    Q2 : BOOL;
    Q3 : BOOL;
END_VAR

VAR
    init : BOOL;
    s0 : TIME;
    s1 : TIME;
    s2 : TIME;
    s3 : TIME;
    tx : TIME;
    c : INT;
END_VAR
(* read system_time *)
tx := DWORD_TO_TIME(T_PLC_MS());

IF NOT init THEN
	init := TRUE;
	s0 := tx - T0;
	s1 := tx - T1;
	s2 := tx - T2;
	s3 := tx - T3;
END_IF;

Q0 := FALSE;
Q1 := FALSE;
Q2 := FALSE;
Q3 :=FALSE;

CASE c OF
	0: 	IF tx - s0 >= T0 THEN
			Q0 := E0;
			s0 := tx;
		END_IF;
		c := 1;
	1: 	IF tx - s1 >= T1 THEN
			Q1 := E1;
			s1 := tx;
		END_IF;
		c := 2;
	2: 	IF tx - s2 >= T2 THEN
			Q2 := E2;
			s2 := tx;
		END_IF;
		c := 3;
	3: 	IF tx - s3 >= T3 THEN
			Q3 := E3;
			s3 := tx;
		END_IF;
		c := 0;
END_CASE;

(* revision history

hm 28. sep. 2008	rev 1.0
	original version

hm	14. mar. 2009	rev 1.1
	removed double assignments

*)
END_FUNCTION_BLOCK

(* ---- SCHEDULER_2.st ---- *)
FUNCTION_BLOCK SCHEDULER_2
VAR_INPUT
    E0 : BOOL;
    E1 : BOOL;
    E2 : BOOL;
    E3 : BOOL;
    C0 : UINT;
    C1 : UINT;
    C2 : UINT;
    C3 : UINT;
    O0 : UINT;
    O1 : UINT;
    O2 : UINT;
    O3 : UINT;
END_VAR

VAR_OUTPUT
    Q0 : BOOL;
    Q1 : BOOL;
    Q2 : BOOL;
    Q3 : BOOL;
END_VAR

VAR
    sx : UINT;
END_VAR
Q0 := E0 AND (sx MOD C0 - O0 = 0);
Q1 := E1 AND (sx MOD C1 - O1 = 0);
Q2 := E2 AND (sx MOD C2 - O2 = 0);
Q3 := E3 AND (sx MOD C3 - O3 = 0);

(* increment cycle counter every cycle *)
sx := sx + 1;

(* revision history
hm 29. sep. 2008		rev 1.0
	original version

*)
END_FUNCTION_BLOCK

(* ---- SEL2_OF_3.st ---- *)
FUNCTION_BLOCK SEL2_OF_3
VAR_INPUT
    IN1 : REAL;
    IN2 : REAL;
    IN3 : REAL;
    D : REAL;
END_VAR

VAR_OUTPUT
    Y : REAL;
    W : INT;
    E : BOOL;
END_VAR

VAR
    D12 : BOOL;
    D23 : BOOL;
    D31 : BOOL;
END_VAR
D12 := ABS(IN1-IN2) <= D;
D23 := ABS(IN2-IN3) <= D;
D31 := ABS(IN3-IN1) <= D;

IF (D12 AND D23) OR (D12 AND D31) OR (D23 AND D31) THEN
	(* all 3 inputs are valid *)
	Y := (IN1 + IN2 + IN3) * 0.333333333333;
	E := FALSE;
	W := 0;
ELSIF D12 THEN
	(* only inut 1 and 2 are valid *)
	Y := (In1 + IN2) * 0.5;
	E := FALSE;
	W := 3;
ELSIF D23 THEN
	(* only inut 2 and 3 are valid *)
	Y := (In2 + IN3) * 0.5;
	E := FALSE;
	W := 1;
ELSIF D31 THEN
	(* only inut 3 and 1 are valid *)
	Y := (In3 + IN1) * 0.5;
	E := FALSE;
	W := 2;
ELSE
	(* no calculation possible *)
	E := TRUE;
	W := 4;
END_IF;

(* revision history
hm	18. may 2008	rev 1.0
	original version

hm	10. mar. 2009	rev 1.1
	improved code
*)
END_FUNCTION_BLOCK

(* ---- SEL2_OF_3B.st ---- *)
FUNCTION_BLOCK SEL2_OF_3B
VAR_INPUT
    IN1 : BOOL;
    IN2 : BOOL;
    IN3 : BOOL;
    TD : TIME;
END_VAR

VAR_OUTPUT
    Q : BOOL;
    W : BOOL;
END_VAR

VAR
    TDEL : TON;
END_VAR
Q := (IN1 AND IN2) OR (IN1 AND IN3) OR (IN2 AND IN3);
TDEL(IN := (in1 XOR in2) OR (in1 XOR in3) OR (in2 XOR in3), PT := TD);
W := TDEL.Q;

(* revision history
hm		19. may 2008	rev 1.0
	original version

*)
END_FUNCTION_BLOCK

(* ---- SELECT_8.st ---- *)
FUNCTION_BLOCK SELECT_8
VAR_INPUT
    E: BOOL;
    SET: BOOL;
    IN: BYTE;
    UP: BOOL;
    DN: BOOL;
    RST: BOOL;
END_VAR

VAR_OUTPUT
    Q0: BOOL;
    Q1: BOOL;
    Q2: BOOL;
    Q3: BOOL;
    Q4: BOOL;
    Q5: BOOL;
    Q6: BOOL;
    Q7: BOOL;
    STATE: INT;
END_VAR

VAR
    last_up: BOOL;
    last_dn: BOOL;
END_VAR
IF rst THEN
	state := 0;
ELSIF set THEN
	state := IN;
ELSIF up AND NOT last_up THEN
	state := inc(state,1,7);
ELSIF dn AND NOT last_dn THEN
	state := inc(state,-1,7);
END_IF;
last_UP := UP;
last_DN := DN;

Q0 := FALSE;
Q1 := FALSE;
Q2 := FALSE;
Q3 := FALSE;
Q4 := FALSE;
Q5 := FALSE;
Q6 := FALSE;
Q7 := FALSE;

IF E THEN
	CASE state OF
		0: Q0 := TRUE;
		1: Q1 := TRUE;
		2: Q2 := TRUE;
		3: Q3 := TRUE;
		4: Q4 := TRUE;
		5: Q5 := TRUE;
		6: Q6 := TRUE;
		7: Q7 := TRUE;
	END_CASE;
END_IF;

(* revision history
hm	16. jan 2008	rev 1.0
	original version

hm	27. feb. 2009	rev 1.1
	renamed input en to e
*)
END_FUNCTION_BLOCK

(* ---- SEQUENCE_4.st ---- *)
FUNCTION_BLOCK SEQUENCE_4
VAR_INPUT
    in0 : BOOL := TRUE;
    in1 : BOOL := TRUE;
    in2 : BOOL := TRUE;
    in3 : BOOL := TRUE;
    start : BOOL;
    rst : BOOL;
    wait0 : TIME;
    delay0 : TIME;
    wait1 : TIME;
    delay1 : TIME;
    wait2 : TIME;
    delay2 : TIME;
    wait3 : TIME;
    delay3 : TIME;
    stop_on_error : BOOL;
END_VAR

VAR_OUTPUT
    Q0 : BOOL;
    Q1 : BOOL;
    Q2 : BOOL;
    Q3 : BOOL;
    QX : BOOL;
    run : BOOL;
    step : INT := -1;
    status : BYTE;
END_VAR

VAR
    last : TIME;
    edge : BOOL;
    tx : TIME;
    init : BOOL;
END_VAR
(* read sps timer *)
tx := DWORD_TO_TIME(T_PLC_MS());

(* initialize on startup *)
IF NOT init THEN
	last := tx;
	init := TRUE;
	status := 110;
END_IF;

(* asynchronous reset *)
IF rst THEN
	step := -1;
	Q0 := 0;
	Q1 := 0;
	Q2 := 0;
	Q3 := 0;
	status := 110;
	run := 0;

(* edge on start input restarts the sequencer *)
ELSIF start AND NOT edge THEN
	step := 0;
	last := tx;
	status := 111;
	Q0 := 0;
	Q1 := 0;
	Q2 := 0;
	Q3 := 0;
	run := 1;
END_IF;
edge := start;

(* check if stop on status is necessary *)
IF status > 0 AND status < 100 AND stop_on_error THEN RETURN; END_IF;

(* sequence is running *)
IF run AND step = 0 THEN
	IF NOT q0 AND in0 AND tx - last <= wait0 THEN
		Q0 := TRUE;
		last := tx;
	ELSIF NOT q0 AND tx - last > wait0 THEN
		status := 1;
		run := FALSE;
	ELSIF q0 AND tx - last >= delay0 THEN
		step := 1;
		last := tx;
	END_IF;
END_IF;
IF run AND step = 1 THEN
	IF NOT q1 AND in1 AND tx - last <= wait1 THEN
		Q0 := FALSE;
		Q1 := TRUE;
		last := tx;
	ELSIF NOT q1 AND Tx - last > wait1 THEN
		status := 2;
		q0 := FALSE;
		run := FALSE;
	ELSIF q1 AND tx - last >= delay1 THEN
		step := 2;
		last := tx;
	END_IF;
END_IF;
IF run AND step = 2 THEN
	IF NOT q2 AND in2 AND tx - last <= wait2 THEN
		Q1 := FALSE;
		Q2 := TRUE;
		last := tx;
	ELSIF NOT q2 AND Tx - last > wait2 THEN
		status := 3;
		q1 := FALSE;
		run := FALSE;
	ELSIF q2 AND tx - last >= delay2 THEN
		step := 3;
		last := tx;
	END_IF;
END_IF;
IF run AND step = 3 THEN
	IF NOT q3 AND in3 AND tx - last <= wait3 THEN
		Q2 := FALSE;
		Q3 := TRUE;
		last := tx;
	ELSIF NOT q3 AND Tx - last > wait3 THEN
		status := 4;
		q2 := FALSE;
		run := FALSE;
	ELSIF q3 AND tx - last >= delay3 THEN
		step := -1;
		q3 := FALSE;
		run := FALSE;
		status := 110;
	END_IF;
END_IF;
QX := q0 OR q1 OR q2 OR q3;

(*
hm 1.10.06		rev 1.1
	corrected delay logic to be after event and not before
	added any output

hm 1.12.06		rev 1.2
	corrected failure in sequence logic.
	added init at startup to prevent from initial error after start.

hm 17.1.2007		rev 1.3
	changed output fault to status for better compatibility with other modules (ESR).
	added stop on error functionality and setup variable
	default for inputs in0..3 is true.
	renamed variable state to step

hm	17.sep 2007	rev 1.4
	replaced time() with T_PLC_MS() for compatibility reasons

hm	13. mar. 2009	rev 1.5
	renamed output any to qx for compatibility resons

*)
END_FUNCTION_BLOCK

(* ---- SEQUENCE_64.st ---- *)
FUNCTION_BLOCK SEQUENCE_64
VAR_INPUT
    START : BOOL;
    SMAX : INT;
    PROG : ARRAY[0..63] OF TIME;
    RST : BOOL;
END_VAR

VAR_OUTPUT
    STATE : INT := -1;
    TRIG : BOOL;
END_VAR

VAR
    tx : TIME;
    edge : BOOL;
    last : TIME;
END_VAR
(* read system timer *)
tx := DWORD_TO_TIME(T_PLC_MS());
TRIG := FALSE;

IF RST THEN
	STATE := -1;

(* start sequence *)
ELSIF START AND NOT edge THEN
	STATE := 0;
	last := tx;
	TRIG := TRUE;

(* sequence generator *)
ELSIF (STATE >= 0) THEN
	IF (tx - last) >= PROG[STATE] THEN
		STATE := INC2(STATE, 1, -1, SMAX);
		last := tx;
		TRIG := TRUE;
	END_IF;
END_IF;

edge := START;

(* revision history
hm	29. jun. 2008
	original version

*)
END_FUNCTION_BLOCK

(* ---- SEQUENCE_8.st ---- *)
FUNCTION_BLOCK SEQUENCE_8
VAR_INPUT
    in0 : BOOL := TRUE;
    in1 : BOOL := TRUE;
    in2 : BOOL := TRUE;
    in3 : BOOL := TRUE;
    in4 : BOOL := TRUE;
    in5 : BOOL := TRUE;
    in6 : BOOL := TRUE;
    in7 : BOOL := TRUE;
    start : BOOL;
    rst : BOOL;
    wait0 : TIME;
    delay0 : TIME;
    wait1 : TIME;
    delay1 : TIME;
    wait2 : TIME;
    delay2 : TIME;
    wait3 : TIME;
    delay3 : TIME;
    wait4 : TIME;
    delay4 : TIME;
    wait5 : TIME;
    delay5 : TIME;
    wait6 : TIME;
    delay6 : TIME;
    wait7 : TIME;
    delay7 : TIME;
    stop_on_error : BOOL;
END_VAR_INPUT

VAR_OUTPUT
    Q0 : BOOL;
    Q1 : BOOL;
    Q2 : BOOL;
    Q3 : BOOL;
    Q4 : BOOL;
    Q5 : BOOL;
    Q6 : BOOL;
    Q7 : BOOL;
    QX : BOOL;
    run : BOOL;
    step : INT := -1;
    status : BYTE;
END_VAR_OUTPUT

VAR_LOCAL
    last : TIME;
    edge : BOOL;
    tx : TIME;
    init : BOOL;
END_VAR_LOCAL
(* read sps timer *)
tx := DWORD_TO_TIME(T_PLC_MS());

(* initialize on startup *)
IF NOT init THEN
	last := tx;
	init := TRUE;
	status := 110;
END_IF;

(* asynchronous reset *)
IF rst THEN
	step := -1;
	Q0 := 0;
	Q1 := 0;
	Q2 := 0;
	Q3 := 0;
	Q4 := 0;
	Q5 := 0;
	Q6 := 0;
	Q7 := 0;
	status := 110;
	run := 0;

(* edge on start input restarts the sequencer *)
ELSIF start AND NOT edge THEN
	step := 0;
	last := tx;
	status := 111;
	Q0 := 0;
	Q1 := 0;
	Q2 := 0;
	Q3 := 0;
	Q4 := 0;
	Q5 := 0;
	Q6 := 0;
	Q7 := 0;
	run := 1;
END_IF;
edge := start;

(* check if stop on error is necessary *)
IF status > 0 AND status < 100 AND stop_on_error THEN RETURN; END_IF;

(* sequence is running *)
IF run AND step = 0 THEN
	IF NOT q0 AND in0 AND tx - last <= wait0 THEN
		Q0 := TRUE;
		last := tx;
	ELSIF NOT q0 AND tx - last > wait0 THEN
		status := 1;
		run := FALSE;
	ELSIF q0 AND tx - last >= delay0 THEN
		step := 1;
		last := tx;
	END_IF;
END_IF;
IF run AND step = 1 THEN
	IF NOT q1 AND in1 AND tx - last <= wait1 THEN
		Q0 := FALSE;
		Q1 := TRUE;
		last := tx;
	ELSIF NOT q1 AND Tx - last > wait1 THEN
		status := 2;
		q0 := FALSE;
		run := FALSE;
	ELSIF q1 AND tx - last >= delay1 THEN
		step := 2;
		last := tx;
	END_IF;
END_IF;
IF run AND step = 2 THEN
	IF NOT q2 AND in2 AND tx - last <= wait2 THEN
		Q1 := FALSE;
		Q2 := TRUE;
		last := tx;
	ELSIF NOT q2 AND Tx - last > wait2 THEN
		status := 3;
		q1 := FALSE;
		run := FALSE;
	ELSIF q2 AND tx - last >= delay2 THEN
		step := 3;
		last := tx;
	END_IF;
END_IF;
IF run AND step = 3 THEN
	IF NOT q3 AND in3 AND tx - last <= wait3 THEN
		Q2 := FALSE;
		Q3 := TRUE;
		last := tx;
	ELSIF NOT q3 AND Tx - last > wait3 THEN
		status := 4;
		q2 := FALSE;
		run := FALSE;
	ELSIF q3 AND tx - last >= delay3 THEN
		step := 4;
		last := tx;
	END_IF;
END_IF;
IF run AND step = 4 THEN
	IF NOT q4 AND in4 AND tx - last <= wait4 THEN
		Q3 := FALSE;
		Q4 := TRUE;
		last := tx;
	ELSIF NOT q4 AND Tx - last > wait4 THEN
		status := 5;
		q3 := FALSE;
		run := FALSE;
	ELSIF q4 AND tx - last >= delay4 THEN
		step := 5;
		last := tx;
	END_IF;
END_IF;
IF run AND step = 5 THEN
	IF NOT q5 AND in5 AND tx - last <= wait5 THEN
		Q4 := FALSE;
		Q5 := TRUE;
		last := tx;
	ELSIF NOT q5 AND Tx - last > wait5 THEN
		status := 6;
		q4 := FALSE;
		run := FALSE;
	ELSIF q5 AND tx - last >= delay5 THEN
		step := 6;
		last := tx;
	END_IF;
END_IF;
IF run AND step = 6 THEN
	IF NOT q6 AND in6 AND tx - last <= wait6 THEN
		Q5 := FALSE;
		Q6 := TRUE;
		last := tx;
	ELSIF NOT q6 AND Tx - last > wait6 THEN
		status := 7;
		q5 := FALSE;
		run := FALSE;
	ELSIF q6 AND tx - last >= delay6 THEN
		step := 7;
		last := tx;
	END_IF;
END_IF;
IF run AND step = 7 THEN
	IF NOT q7 AND in7 AND tx - last <= wait7 THEN
		Q6 := FALSE;
		Q7 := TRUE;
		last := tx;
	ELSIF NOT q7 AND Tx - last > wait7 THEN
		status := 8;
		q6 := FALSE;
		run := FALSE;
	ELSIF q7 AND tx - last >= delay7 THEN
		step := -1;
		Q7 := FALSE;
		Run := FALSE;
		status := 110;
	END_IF;
END_IF;
QX := q0 OR q1 OR q2 OR q3 OR q4 OR q5 OR q6 OR q7;

(*
hm 1.10.06		rev 1.1
	corrected delay logic to be after event and not before
	added any output

hm 1.12.06		rev 1.2
	corrected failure in sequence logic.
	added init at startup to prevent from initial statuss after start.

hm 17.1.2007		rev 1.3
	changed output fault to status for better compatibility with other modules (ESR)
	added stop on error functionality and setup variable
	default for inputs in0..7 is true.
	renames variable state to step

hm	17.sep 2007	rev 1.4
	replaced time() with T_PLC_MS() for compatibility reasons

hm	13. mar. 2009	rev 1.5
	renamed output any to qx for compatibility resons

*)
END_FUNCTION_BLOCK

(* ---- SH.st ---- *)
FUNCTION_BLOCK SH
VAR_INPUT
    in : REAL;    (* Input Real Variable *)
    CLK : BOOL;   (* Clock Input Variable *)
END_VAR

VAR_OUTPUT
    out : REAL;   (* Output Real Variable *)
    trig : BOOL;  (* Output BOOL Variable *)
END_VAR

VAR
    edge : BOOL;  (* Local BOOL Variable *)
END_VAR
IF clk AND NOT edge THEN
	out := in;
	trig := TRUE;
ELSE;
	trig := FALSE;
END_IF;
edge := clk;

(* revision history

hm 16.1.2007	rev 1.1
	added trig output

*)
END_FUNCTION_BLOCK

(* ---- SH_1.st ---- *)
FUNCTION_BLOCK SH_1
VAR_INPUT
    in : REAL;
    PT : TIME;
END_VAR

VAR_OUTPUT
    out : REAL;
    Trig : BOOL;
END_VAR

VAR
    last : TIME;
    tx : TIME;
END_VAR
(* read system time *)
tx := DWORD_TO_TIME(T_PLC_MS());

IF tx - last >= PT THEN
	last := tx;
	out := in;
	trig := TRUE;
ELSE
	trig := FALSE;
END_IF;

(* revision history

HM	6.1.2007	rev 1.1
	added trig output

HM	17.9.2007	rev 1.2
	replaced time() with T_PLC_MS() for compatibility reasons
*)
END_FUNCTION_BLOCK

(* ---- SH_2.st ---- *)
FUNCTION_BLOCK SH_2
VAR_INPUT
    in : REAL;
    PT : TIME;
    N : INT := 16;
    disc : INT;
END_VAR

VAR_OUTPUT
    out : REAL;
    trig : BOOL;
    avg : REAL;
    high : REAL;
    low : REAL;
END_VAR

VAR
    M : INT;
    buf : ARRAY[0..15] OF REAL;
    buf2 : ARRAY[0..15] OF REAL;
    last : TIME;
    i : INT;
    start : INT;
    temp : REAL;
    stop : INT;
    tx : TIME;
    d2 : INT;
END_VAR
(* read system time *)
tx := DWORD_TO_TIME(T_PLC_MS());
d2 := SHR(disc,1);

IF tx - last >= PT THEN
	last := tx;
	trig := TRUE;

	(* limit M to 0..16 *)
	M := LIMIT(1,N,16);

	(* edge detected lets take the sample *)
	FOR i := M - 1 TO 1 BY -1 DO buf2[i] := buf2[i-1]; END_FOR;
	buf2[0] := in;
	out := in;
	buf := buf2;

	(* sort the ARRAY lowest value AT 0 *)
	FOR start := 0 TO M - 2 DO
		FOR i := start+1 TO M - 1 DO
			IF buf[start] > buf[i] THEN
				temp := buf[start];
				buf[start] := buf[i];
				buf[i] := temp;
			END_IF;
		END_FOR;
	END_FOR;

	(* any calculation with the samples is here *)
	stop := M - 1 - d2;
	start := d2;
	IF NOT even(disc) THEN start := start + 1; END_IF;
	avg := 0;
	FOR i := start TO stop DO avg := avg + buf[i]; END_FOR;
	avg := avg / INT_TO_REAL(stop - start +1);
	low := buf[start];
	high := buf[stop];
ELSE
	Trig := FALSE;
END_IF;

(* revision history
hm 20. jan. 2007	rev 1.1
	added input N to specify the amout of samples for average and high low calculations
	added trig output

hm 10. sep. 2007 	rev 1.2
	an error would be generated if N was set to 0, now n is forced to1 if set to 0.
	index was out of array.

hm	17. sep. 2007	rev 1.3
	replaced time() with t_plc_ms() for compatibility reasons

hm	6. jan. 2008	rev 1.4
	improved performance

hm	14. jun. 2008	rev 1.5
	set default for input N = 16

hm	10. mar. 2009	rev 1.6
	added type conversion for compatibility reasons

*)
END_FUNCTION_BLOCK

(* ---- SH_T.st ---- *)
FUNCTION_BLOCK SH_T
VAR_INPUT
    IN : REAL;
    E : BOOL;
END_VAR

VAR_OUTPUT
    OUT : REAL;
END_VAR
IF E THEN out := in; END_IF;

(* revision history
hm	1. sep. 2006	rev 1.0
	original version

hm	18. oct. 2008	rev 1.1
	changed input en to e for compatibility reasons

*)
END_FUNCTION_BLOCK

(* ---- SHR_4E.st ---- *)
FUNCTION_BLOCK SHR_4E
VAR_INPUT
    SET : BOOL;
    D0 : BOOL;
    CLK : BOOL;
    RST : BOOL;
END_VAR

VAR_OUTPUT
    Q0 : BOOL;
    Q1 : BOOL;
    Q2 : BOOL;
    Q3 : BOOL;
END_VAR

VAR
    trig : R_TRIG;
END_VAR
(* trig.Q signals a rising edge on clk *)
trig(clk := clk);

IF set OR rst THEN
	Q0 := NOT rst;
	Q1 := Q0;
	Q2 := Q0;
	Q3 := Q0;
ELSIF trig.Q THEN
	Q3 := Q2;
	Q2 := Q1;
	Q1 := Q0;
	Q0 := D0;
END_IF;

(* revision history
hm	4. aug. 2006	rev 1.0
	original version

hm	25. oct. 2008	rev 1.1
	optimized code

*)
END_FUNCTION_BLOCK

(* ---- SHR_4UDE.st ---- *)
FUNCTION_BLOCK SHR_4UDE
VAR_INPUT
    SET : BOOL;
    D0 : BOOL;
    D3 : BOOL;
    CLK : BOOL;
    DN : BOOL;
    RST : BOOL;
END_VAR

VAR_OUTPUT
    Q0 : BOOL;
    Q1 : BOOL;
    Q2 : BOOL;
    Q3 : BOOL;
END_VAR

VAR
    trig : R_TRIG;
END_VAR
(* trig.Q signals a rising edge on clk *)
trig(clk := clk);

IF set OR rst THEN
	Q0 := NOT RST;
	Q1 := Q0;
	Q2 := Q0;
	Q3 := Q0;
ELSIF trig.Q THEN
	IF dn THEN
		Q0 := Q1;
		Q1 := Q2;
		Q2 := Q3;
		Q3 := D3;
	ELSE
		Q3 := Q2;
		Q2 := Q1;
		Q1 := Q0;
		Q0 := D0;
	END_IF;
END_IF;

(* revision history
hm	4. aug. 2006	rev 1.0
	original version

hm	25. oct. 2008	rev 1.1
	optimized code

hm	14. mar. 2009	rev 1.2
	removed double assignments

*)
END_FUNCTION_BLOCK

(* ---- SHR_8PLE.st ---- *)
FUNCTION_BLOCK SHR_8PLE
VAR_INPUT
    Din : BOOL;
    Dload : BYTE;
    CLK : BOOL;
    UP : BOOL := TRUE; // Initial Value = 1
    load : BOOL;
    RST : BOOL;
END_VAR

VAR_OUTPUT
    DOut : BOOL;
END_VAR

VAR
    edge : BOOL := TRUE; // Initial Value = 1
    register : BYTE;
END_VAR
(* flankenerkennung clk wird high und edge war high reset ist nicht aktiv und set ist nicht aktiv *)
IF CLK AND edge AND NOT rst THEN
	edge := FALSE;	(* flanke wurde erkannt und weitere flankenerkennung wird verhindert bis edge wieder true ist *)
	(* hier ist der code für das flankenevent *)
	IF UP THEN						(*shift up *)
		register := SHL(register,1);
		register.0 := Din;
		Dout := register.7;
	ELSE								(* shift down *);
		register := SHR(register,1);
		register.7 := Din;
		Dout := register.0;
	END_IF;
	IF load THEN							(* the byte on Din will be loaded if load = true *)
		register := Dload;
		IF up THEN Dout := register.7; ELSE Dout := register.0; END_IF;
	END_IF;
END_IF;
IF NOT clk THEN edge := TRUE; END_IF;	(* sobald clk wieder low wird warten auf nächste flanke *)
IF rst THEN									(* wenn reset aktiv dann ausgang rücksetzen *)
	register := 0;
	Dout := FALSE;
END_IF;
END_FUNCTION_BLOCK

(* ---- SHR_8UDE.st ---- *)
FUNCTION_BLOCK SHR_8UDE
VAR_INPUT
    SET : BOOL;
    D0 : BOOL;
    D7 : BOOL;
    CLK : BOOL;
    DN : BOOL;
    RST : BOOL;
END_VAR

VAR_OUTPUT
    Q0 : BOOL;
    Q1 : BOOL;
    Q2 : BOOL;
    Q3 : BOOL;
    Q4 : BOOL;
    Q5 : BOOL;
    Q6 : BOOL;
    Q7 : BOOL;
END_VAR

VAR
    trig : R_TRIG;
END_VAR
(* trig.Q signals a rising edge on clk *)
trig(clk := clk);

IF set OR rst THEN
	Q0 := NOT RST;
	Q1 := Q0;
	Q2 := Q0;
	Q3 := Q0;
	Q4 := Q0;
	Q5 := Q0;
	Q6 := Q0;
	Q7 := Q0;
ELSIF trig.Q THEN
	IF dn THEN
		Q0 := Q1;
		Q1 := Q2;
		Q2 := Q3;
		Q3 := Q4;
		Q4 := Q5;
		Q5 := Q6;
		Q6 := Q7;
		Q7 := D7;
	ELSE
		Q7 := Q6;
		Q6 := Q5;
		Q5 := Q4;
		Q4 := Q3;
		Q3 := Q2;
		Q2 := Q1;
		Q1 := Q0;
		Q0 := D0;
	END_IF;
END_IF;

(* revision history
hm	4. aug. 2006	rev 1.0
	original version

hm	25. oct. 2008	rev 1.1
	optimized code

hm	14. mar. 2009	rev 1.2
	removed double assignments

*)
END_FUNCTION_BLOCK

(* ---- SIGNAL.st ---- *)
FUNCTION_BLOCK SIGNAL
VAR_INPUT
    IN : BOOL;
    SIG : BYTE;
    TS : TIME;
END_VAR

VAR_OUTPUT
    Q : BOOL;
END_VAR

VAR
    tx : DWORD;
    step : BYTE;
END_VAR

VAR CONSTANT
    one : BYTE := 1;
END_VAR
IF in THEN
	(* an alarm is present read system time first *)
	tx := T_PLC_MS();
	(* calculate the step counter which is the lowest 3 bits of (time / ts) *)
	IF ts > t#0s THEN
		step := DWORD_TO_BYTE(tx / TIME_TO_DWORD(ts) AND 16#0000_0007);
	ELSE
		step := DWORD_TO_BYTE(SHR(tx,7) AND 16#0000_0007);
	END_IF;
	(* convert the value 0-7 in step into one bit only (bit 0-7) *)
	step := SHL(one,step);
	(* generate the output signal *)
	Q := (step AND sig) > 0;
ELSE
	Q := FALSE;
END_IF;

(* revision history
hm	13.12.2007		rev 1.0
	original version

*)
END_FUNCTION_BLOCK

(* ---- SIGNAL_4.st ---- *)
FUNCTION_BLOCK SIGNAL_4
VAR_INPUT
    IN1 : BOOL;
    IN2 : BOOL;
    IN3 : BOOL;
    IN4 : BOOL;
    TS : TIME;
    S1 : BYTE := 16#FF;  // Initial value set as 2#11111111
    S2 : BYTE := 16#F0;  // Initial value set as 2#11110000
    S3 : BYTE := 16#AA;  // Initial value set as 2#10101010
    S4 : BYTE := 16#A0;  // Initial value set as 2#10100000
END_VAR

VAR_OUTPUT
    Q : BOOL;
END_VAR

VAR
    sig : SIGNAL;  // Local variable of derived type SIGNAL
END_VAR
(* an alarm is present read system time first *)
(* check if an alarm is present if yes set sig to the alarm pattern otherwise exit the routine *)
IF in1 THEN
	sig(in := TRUE, sig := s1, TS := TS);
ELSIF in2 THEN
	sig(in := TRUE, sig := s2, TS := TS);
ELSIF in3 THEN
	sig(in := TRUE, sig := s3, TS := TS);
ELSIF in4 THEN
	sig(in := TRUE, sig := s4, TS := TS);
ELSE
	sig(in := FALSE);
END_IF;

(* set the output *)
Q := sig.Q;

(* revision history
hm	13.12.2007		rev 1.0
	original version

*)
END_FUNCTION_BLOCK

(* ---- SPEED.st ---- *)
FUNCTION_BLOCK SPEED
VAR_INPUT
    ms : REAL;
    kmh : REAL;
    kn : REAL;
    mh : REAL;
END_VAR

VAR_OUTPUT
    Yms : REAL;
    Ykmh : REAL;
    Ykn : REAL;
    Ymh : REAL;
END_VAR
Yms := ms +
		kmh * 0.27777777777778 +
		kn * 0.5144444 +
		mh * 0.44704;
Ykmh := Yms * 3.6;
Ykn := Yms * 1.94384466037535;
Ymh := Yms * 2.23693629205440;

(*
Geschwindigkeit Meter durch Sekunde m/s 1 m/s = 3,6 km/h
km durch (pro) Stunde, nicht „Stundenkilometer“ verwenden
Knoten kn 1 kn = 1 sm/h = 0,5144 m/s

*)

(* revision history
hm	27. mar. 2009	rev 1.0
	original version

hm	11. mar. 2009	rev 1.1
	improved code

*)
END_FUNCTION_BLOCK

(* ---- SRAMP.st ---- *)
FUNCTION_BLOCK SRAMP
VAR_INPUT
    X           : REAL;
    A_UP        : REAL;
    A_DN        : REAL;
    VU_MAX      : REAL;
    VD_MAX      : REAL;
    LIMIT_HIGH  : REAL;
    LIMIT_LOW   : REAL;
    RST         : BOOL;
END_VAR

VAR_OUTPUT
    Y           : REAL;
    V           : REAL;
END_VAR

VAR
    cycle_time  : TC_S;
    init        : BOOL;
END_VAR
(* read the system_time in microseconds *)
cycle_time();

(* assure range of inputs *)
A_up := MAX(0.0, A_UP);
A_dn := MIN(0.0, A_dn);
VU_max := MAX(0.0, VU_max);
VD_max := MIN(0.0, VD_MAX);

(* calculate the output offset *)
IF rst OR NOT init THEN
	init := TRUE;
	Y := 0.0;
	V := 0.0;
ELSIF X = Y THEN
	v := 0.0;
ELSIF X > Y THEN
	(* output is too low >> ramp up and brake at the end *)
	(* accelerate the speed and limit to vu_max *)
	v := MIN(v + A_UP * cycle_time.TC, vu_max);
	(* calculate the max speed to be able to brake and select the lowest *)
	v := MIN(SQRT((Y-X) * 2.0 * A_DN), v);
	(* calculate the output and obey limits *)
	y := LIMIT(limit_low, y + MIN(v * cycle_time.TC, X-Y), limit_high);
ELSIF X < Y THEN
	(* output is too high >> ramp dn and brake at the end *)
	(* accelerate the speed and limit to vd_max *)
	v := MAX(v + A_DN * cycle_time.TC, vd_max);
	(* calculate the max speed to be able to brake and select the lowest *)
	v := MAX(-SQRT((Y-X) * 2.0 * A_UP), v);
	(* calculate the output and obey limits *)
	y := LIMIT(limit_low, y + MAX(v * cycle_time.TC, X-Y), limit_high);
END_IF;

(* revision history
hm	13. mar. 2008	rev 1.0
	original version

hm	11. mar. 2009	rev 1.1
	real constants updated to new systax using dot

*)
END_FUNCTION_BLOCK

(* ---- STACK_16.st ---- *)
FUNCTION_BLOCK STACK_16
VAR_INPUT
    Din : DWORD;
    E : BOOL := TRUE;
    RD : BOOL;
    WD : BOOL;
    RST : BOOL;
END_VAR

VAR_OUTPUT
    Dout : DWORD;
    EMPTY : BOOL := TRUE;
    FULL : BOOL;
END_VAR

VAR
    stack : ARRAY[0..n] OF DWORD;
    pt : INT;
END_VAR

VAR CONSTANT
    n : INT := 15; (* changing this value will change the number of stored elements in the fifo *)
END_VAR
IF RST THEN
	(* asynchronous reset for the fifo *)
	pt := 0;
	EMPTY := TRUE;
	FULL := FALSE;
	Dout := 0;
ELSIF E THEN
	IF NOT EMPTY AND RD THEN
		(* read one element *)
		pt := pt - 1;
		Dout := stack[pt];
		EMPTY := pt = 0;
		FULL := FALSE;
	END_IF;
	IF NOT FULL AND WD THEN
		(* write one element *)
		stack[pt] := Din;
		pt := pt + 1;
		FULL := pt > n;
		EMPTY := FALSE;
	END_IF;
END_IF;

(* revision history
hm	4. aug. 2006	rev 1.0
	original version

hm	19. feb 2008	rev 1.1
	performance improvements

hm	17. oct. 2008	rev 1.2
	deleted unnecessary init with 0

hm	27. oct. 2008	rev 1.3
	optimized performance

hm	25. jul 2009	rev 2.0
	changed inputs to allow simultsaneous read and write
*)
END_FUNCTION_BLOCK
